LIN {X 0,Y 480.885,Z 595.896,A -85,B 0,C 180,E1 22639.921,E2 22639.921} C_VEL
LIN {X 0,Y 480.883,Z 595.897,A -85,B 0,C 180,E1 22636.346,E2 22636.346} C_VEL
LIN {X 0,Y 480.836,Z 595.897,A -85,B 0,C 180,E1 22632.842,E2 22632.842} C_VEL
LIN {X 0,Y 480.862,Z 595.898,A -85,B 0,C 180,E1 22629.331,E2 22629.331} C_VEL
LIN {X 0,Y 480.868,Z 596.139,A -85,B 0,C 180,E1 22626.726,E2 22626.726} C_VEL
LIN {X 0,Y 487.982,Z 616.092,A -85,B 0,C 180,E1 22624.296,E2 22624.296} C_VEL
LIN {X 0,Y 491.181,Z 625.758,A -85,B 0,C 180,E1 22623.202,E2 22623.202} C_VEL
LIN {X 0,Y 488.684,Z 670.223,A -85,B 0,C 180,E1 22619.477,E2 22619.477} C_VEL
LIN {X 0,Y 487.647,Z 692.767,A -85,B 0,C 180,E1 22617.655,E2 22617.655} C_VEL
LIN {X 0,Y 489.758,Z 709.939,A -85,B 0,C 180,E1 22617.279,E2 22617.279} C_VEL
LIN {X 0,Y 487.922,Z 898.558,A -85,B 0,C 180,E1 22614.449,E2 22614.449} C_VEL
LIN {X 0,Y 487.32,Z 917.588,A -85,B 0,C 180,E1 22613.95,E2 22613.95} C_VEL
LIN {X 0,Y 486.57,Z 936.141,A -85,B 0,C 180,E1 22613.238,E2 22613.238} C_VEL
LIN {X 0,Y 485.716,Z 953.916,A -85,B 0,C 180,E1 22612.33,E2 22612.33} C_VEL
LIN {X 0,Y 484.717,Z 971.45,A -85,B 0,C 180,E1 22611.193,E2 22611.193} C_VEL
LIN {X 0,Y 483.784,Z 987.738,A -85,B 0,C 180,E1 22609.886,E2 22609.886} C_VEL
LIN {X 0,Y 482.865,Z 1003.139,A -85,B 0,C 180,E1 22608.388,E2 22608.388} C_VEL
LIN {X 0,Y 482.045,Z 1017.074,A -85,B 0,C 180,E1 22606.757,E2 22606.757} C_VEL
LIN {X 0,Y 481.368,Z 1029.509,A -85,B 0,C 180,E1 22605.014,E2 22605.014} C_VEL
LIN {X 0,Y 480.819,Z 1040.852,A -85,B 0,C 180,E1 22603.101,E2 22603.101} C_VEL
LIN {X 0,Y 480.43,Z 1050.286,A -85,B 0,C 180,E1 22601.16,E2 22601.16} C_VEL
LIN {X 0,Y 480.175,Z 1058.316,A -85,B 0,C 180,E1 22599.106,E2 22599.106} C_VEL
LIN {X 0,Y 480.025,Z 1064.517,A -85,B 0,C 180,E1 22597.059,E2 22597.059} C_VEL
LIN {X 0,Y 479.944,Z 1069.266,A -85,B 0,C 180,E1 22594.9,E2 22594.9} C_VEL
LIN {X 0,Y 479.92,Z 1072.251,A -85,B 0,C 180,E1 22592.747,E2 22592.747} C_VEL
LIN {X 0,Y 479.918,Z 1073.547,A -85,B 0,C 180,E1 22590.597,E2 22590.597} C_VEL
LIN {X 0,Y 479.919,Z 1073.107,A -85,B 0,C 180,E1 22588.329,E2 22588.329} C_VEL
LIN {X 0,Y 479.933,Z 1070.8,A -85,B 0,C 180,E1 22586.058,E2 22586.058} C_VEL
LIN {X 0,Y 479.981,Z 1066.842,A -85,B 0,C 180,E1 22583.902,E2 22583.902} C_VEL
LIN {X 0,Y 480.102,Z 1061.058,A -85,B 0,C 180,E1 22581.738,E2 22581.738} C_VEL
LIN {X 0,Y 480.326,Z 1053.297,A -85,B 0,C 180,E1 22579.566,E2 22579.566} C_VEL
LIN {X 0,Y 480.68,Z 1043.941,A -85,B 0,C 180,E1 22577.507,E2 22577.507} C_VEL
LIN {X 0,Y 481.187,Z 1033.056,A -85,B 0,C 180,E1 22575.561,E2 22575.561} C_VEL
LIN {X 0,Y 481.832,Z 1020.659,A -85,B 0,C 180,E1 22573.732,E2 22573.732} C_VEL
LIN {X 0,Y 482.639,Z 1006.709,A -85,B 0,C 180,E1 22572.021,E2 22572.021} C_VEL
LIN {X 0,Y 483.522,Z 991.701,A -85,B 0,C 180,E1 22570.491,E2 22570.491} C_VEL
LIN {X 0,Y 484.44,Z 975.717,A -85,B 0,C 180,E1 22569.143,E2 22569.143} C_VEL
LIN {X 0,Y 485.421,Z 958.353,A -85,B 0,C 180,E1 22567.956,E2 22567.956} C_VEL
LIN {X 0,Y 486.296,Z 940.865,A -85,B 0,C 180,E1 22567.005,E2 22567.005} C_VEL
LIN {X 0,Y 487.081,Z 922.417,A -85,B 0,C 180,E1 22566.239,E2 22566.239} C_VEL
LIN {X 0,Y 487.711,Z 903.808,A -85,B 0,C 180,E1 22565.693,E2 22565.693} C_VEL
LIN {X 0,Y 488.08,Z 882.284,A -85,B 0,C 180,E1 22565.306,E2 22565.306} C_VEL
LIN {X 0,Y 489.493,Z 707.074,A -85,B 0,C 180,E1 22562.699,E2 22562.699} C_VEL
LIN {X 0,Y 487.571,Z 692.581,A -85,B 0,C 180,E1 22562.362,E2 22562.362} C_VEL
LIN {X 0,Y 489.651,Z 650.462,A -85,B 0,C 180,E1 22558.894,E2 22558.894} C_VEL
LIN {X 0,Y 491.217,Z 625.654,A -85,B 0,C 180,E1 22556.781,E2 22556.781} C_VEL
LIN {X 0,Y 484.613,Z 606.437,A -85,B 0,C 180,E1 22554.482,E2 22554.482} C_VEL
LIN {X 0,Y 480.883,Z 596.216,A -85,B 0,C 180,E1 22553.128,E2 22553.128} C_VEL
LIN {X 0,Y 480.846,Z 595.905,A -85,B 0,C 180,E1 22551.621,E2 22551.621} C_VEL
LIN {X 0,Y 480.897,Z 595.893,A -85,B 0,C 180,E1 22548.133,E2 22548.133} C_VEL
LIN {X 0,Y 480.845,Z 595.899,A -85,B 0,C 180,E1 22544.654,E2 22544.654} C_VEL
LIN {X 0,Y 480.838,Z 595.9,A -85,B 0,C 180,E1 22541.078,E2 22541.078} C_VEL
LIN {X 0,Y 480.897,Z 595.89,A -85,B 0,C 180,E1 22537.681,E2 22537.681} C_VEL
LIN {X 0,Y 480.854,Z 595.896,A -85,B 0,C 180,E1 22534.149,E2 22534.149} C_VEL
LIN {X 0,Y 480.837,Z 595.9,A -85,B 0,C 180,E1 22530.585,E2 22530.585} C_VEL
LIN {X 0,Y 480.89,Z 595.889,A -85,B 0,C 180,E1 22527.14,E2 22527.14} C_VEL
LIN {X 0,Y 480.863,Z 595.889,A -85,B 0,C 180,E1 22523.66,E2 22523.66} C_VEL
LIN {X 0,Y 480.841,Z 595.894,A -85,B 0,C 180,E1 22520.193,E2 22520.193} C_VEL
LIN {X 0,Y 480.885,Z 595.899,A -85,B 0,C 180,E1 22516.674,E2 22516.674} C_VEL
LIN {X 0,Y 480.867,Z 595.89,A -85,B 0,C 180,E1 22513.222,E2 22513.222} C_VEL
LIN {X 0,Y 480.843,Z 595.886,A -85,B 0,C 180,E1 22509.696,E2 22509.696} C_VEL
LIN {X 0,Y 480.881,Z 595.895,A -85,B 0,C 180,E1 22506.207,E2 22506.207} C_VEL
LIN {X 0,Y 480.882,Z 595.893,A -85,B 0,C 180,E1 22502.622,E2 22502.622} C_VEL
LIN {X 0,Y 480.848,Z 595.892,A -85,B 0,C 180,E1 22499.166,E2 22499.166} C_VEL
LIN {X 0,Y 480.87,Z 595.888,A -85,B 0,C 180,E1 22495.587,E2 22495.587} C_VEL
LIN {X 0,Y 480.896,Z 595.896,A -85,B 0,C 180,E1 22491.992,E2 22491.992} C_VEL
LIN {X 0,Y 480.859,Z 595.897,A -85,B 0,C 180,E1 22488.485,E2 22488.485} C_VEL
LIN {X 0,Y 480.855,Z 595.899,A -85,B 0,C 180,E1 22484.811,E2 22484.811} C_VEL
LIN {X 0,Y 480.892,Z 595.895,A -85,B 0,C 180,E1 22481.325,E2 22481.325} C_VEL
LIN {X 0,Y 480.886,Z 595.895,A -85,B 0,C 180,E1 22477.706,E2 22477.706} C_VEL
LIN {X 0,Y 480.86,Z 595.897,A -85,B 0,C 180,E1 22474.109,E2 22474.109} C_VEL
LIN {X 0,Y 480.875,Z 595.894,A -85,B 0,C 180,E1 22470.476,E2 22470.476} C_VEL
LIN {X 0,Y 480.893,Z 595.897,A -85,B 0,C 180,E1 22466.85,E2 22466.85} C_VEL
LIN {X 0,Y 480.882,Z 595.898,A -85,B 0,C 180,E1 22463.214,E2 22463.214} C_VEL
LIN {X 0,Y 480.94,Z 596.225,A -85,B 0,C 180,E1 22462.577,E2 22462.577} C_VEL
LIN {X 0,Y 485.634,Z 612.199,A -85,B 0,C 180,E1 22459.877,E2 22459.877} C_VEL
LIN {X 0,Y 487.628,Z 620.026,A -85,B 0,C 180,E1 22458.631,E2 22458.631} C_VEL
LIN {X 0,Y 485.867,Z 648.971,A -85,B 0,C 180,E1 22454.807,E2 22454.807} C_VEL
LIN {X 0,Y 484.335,Z 678.124,A -85,B 0,C 180,E1 22451.032,E2 22451.032} C_VEL
LIN {X 0,Y 483.003,Z 708.393,A -85,B 0,C 180,E1 22447.182,E2 22447.182} C_VEL
LIN {X 0,Y 483.679,Z 712.593,A -85,B 0,C 180,E1 22447.023,E2 22447.023} C_VEL
LIN {X 0,Y 484.283,Z 715.766,A -85,B 0,C 180,E1 22446.942,E2 22446.942} C_VEL
LIN {X 0,Y 484.176,Z 720.144,A -85,B 0,C 180,E1 22446.877,E2 22446.877} C_VEL
LIN {X 0,Y 481.662,Z 727.25,A -85,B 0,C 180,E1 22446.89,E2 22446.89} C_VEL
LIN {X 0,Y 478.477,Z 735.14,A -85,B 0,C 180,E1 22446.924,E2 22446.924} C_VEL
LIN {X 0,Y 477.919,Z 738.903,A -85,B 0,C 180,E1 22446.892,E2 22446.892} C_VEL
LIN {X 0,Y 476.905,Z 825.971,A -85,B 0,C 180,E1 22445.471,E2 22445.471} C_VEL
LIN {X 0,Y 476.579,Z 841.641,A -85,B 0,C 180,E1 22444.979,E2 22444.979} C_VEL
LIN {X 0,Y 476.066,Z 856.592,A -85,B 0,C 180,E1 22444.254,E2 22444.254} C_VEL
LIN {X 0,Y 475.466,Z 870.004,A -85,B 0,C 180,E1 22443.361,E2 22443.361} C_VEL
LIN {X 0,Y 474.82,Z 882.624,A -85,B 0,C 180,E1 22442.265,E2 22442.265} C_VEL
LIN {X 0,Y 474.198,Z 894.207,A -85,B 0,C 180,E1 22440.963,E2 22440.963} C_VEL
LIN {X 0,Y 473.624,Z 903.957,A -85,B 0,C 180,E1 22439.568,E2 22439.568} C_VEL
LIN {X 0,Y 473.133,Z 912.641,A -85,B 0,C 180,E1 22437.979,E2 22437.979} C_VEL
LIN {X 0,Y 472.77,Z 919.786,A -85,B 0,C 180,E1 22436.232,E2 22436.232} C_VEL
LIN {X 0,Y 472.546,Z 924.839,A -85,B 0,C 180,E1 22434.501,E2 22434.501} C_VEL
LIN {X 0,Y 472.426,Z 928.327,A -85,B 0,C 180,E1 22432.655,E2 22432.655} C_VEL
LIN {X 0,Y 472.374,Z 930.028,A -85,B 0,C 180,E1 22430.679,E2 22430.679} C_VEL
LIN {X 0,Y 472.37,Z 929.733,A -85,B 0,C 180,E1 22428.768,E2 22428.768} C_VEL
LIN {X 0,Y 472.42,Z 927.698,A -85,B 0,C 180,E1 22426.933,E2 22426.933} C_VEL
LIN {X 0,Y 472.546,Z 923.813,A -85,B 0,C 180,E1 22425.085,E2 22425.085} C_VEL
LIN {X 0,Y 472.773,Z 918.177,A -85,B 0,C 180,E1 22423.328,E2 22423.328} C_VEL
LIN {X 0,Y 473.116,Z 911.095,A -85,B 0,C 180,E1 22421.705,E2 22421.705} C_VEL
LIN {X 0,Y 473.581,Z 902.634,A -85,B 0,C 180,E1 22420.215,E2 22420.215} C_VEL
LIN {X 0,Y 474.15,Z 892.288,A -85,B 0,C 180,E1 22418.794,E2 22418.794} C_VEL
LIN {X 0,Y 474.727,Z 880.939,A -85,B 0,C 180,E1 22417.564,E2 22417.564} C_VEL
LIN {X 0,Y 475.391,Z 867.786,A -85,B 0,C 180,E1 22416.461,E2 22416.461} C_VEL
LIN {X 0,Y 475.944,Z 854.292,A -85,B 0,C 180,E1 22415.606,E2 22415.606} C_VEL
LIN {X 0,Y 476.403,Z 839.891,A -85,B 0,C 180,E1 22414.94,E2 22414.94} C_VEL
LIN {X 0,Y 476.721,Z 823.999,A -85,B 0,C 180,E1 22414.466,E2 22414.466} C_VEL
LIN {X 0,Y 477.568,Z 722.274,A -85,B 0,C 180,E1 22412.847,E2 22412.847} C_VEL
LIN {X 0,Y 475.196,Z 708.93,A -85,B 0,C 180,E1 22412.502,E2 22412.502} C_VEL
LIN {X 0,Y 476.348,Z 681.616,A -85,B 0,C 180,E1 22409.038,E2 22409.038} C_VEL
LIN {X 0,Y 477.85,Z 653.013,A -85,B 0,C 180,E1 22405.319,E2 22405.319} C_VEL
LIN {X 0,Y 479.563,Z 623.964,A -85,B 0,C 180,E1 22401.487,E2 22401.487} C_VEL
LIN {X 0,Y 479.484,Z 620.492,A -85,B 0,C 180,E1 22401.002,E2 22401.002} C_VEL
LIN {X 0,Y 474.295,Z 601.706,A -85,B 0,C 180,E1 22398.004,E2 22398.004} C_VEL
LIN {X 0,Y 472.958,Z 596.977,A -85,B 0,C 180,E1 22397.175,E2 22397.175} C_VEL
LIN {X 0,Y 472.94,Z 596.887,A -85,B 0,C 180,E1 22393.543,E2 22393.543} C_VEL
LIN {X 0,Y 472.936,Z 596.88,A -85,B 0,C 180,E1 22389.833,E2 22389.833} C_VEL
LIN {X 0,Y 472.947,Z 596.853,A -85,B 0,C 180,E1 22386.265,E2 22386.265} C_VEL
LIN {X 0,Y 472.949,Z 596.886,A -85,B 0,C 180,E1 22382.556,E2 22382.556} C_VEL
LIN {X 0,Y 472.931,Z 596.851,A -85,B 0,C 180,E1 22378.945,E2 22378.945} C_VEL
LIN {X 0,Y 472.936,Z 596.883,A -85,B 0,C 180,E1 22375.327,E2 22375.327} C_VEL
LIN {X 0,Y 472.953,Z 596.879,A -85,B 0,C 180,E1 22371.659,E2 22371.659} C_VEL
LIN {X 0,Y 472.949,Z 596.877,A -85,B 0,C 180,E1 22368.082,E2 22368.082} C_VEL
LIN {X 0,Y 472.931,Z 596.885,A -85,B 0,C 180,E1 22364.411,E2 22364.411} C_VEL
LIN {X 0,Y 472.933,Z 596.866,A -85,B 0,C 180,E1 22360.79,E2 22360.79} C_VEL
LIN {X 0,Y 472.952,Z 596.882,A -85,B 0,C 180,E1 22357.202,E2 22357.202} C_VEL
LIN {X 0,Y 472.952,Z 596.869,A -85,B 0,C 180,E1 22353.489,E2 22353.489} C_VEL
LIN {X 0,Y 472.92,Z 596.886,A -85,B 0,C 180,E1 22349.906,E2 22349.906} C_VEL
LIN {X 0,Y 472.934,Z 596.864,A -85,B 0,C 180,E1 22346.309,E2 22346.309} C_VEL
LIN {X 0,Y 472.955,Z 596.884,A -85,B 0,C 180,E1 22342.761,E2 22342.761} C_VEL
LIN {X 0,Y 472.931,Z 596.876,A -85,B 0,C 180,E1 22339.129,E2 22339.129} C_VEL
LIN {X 0,Y 472.916,Z 596.876,A -85,B 0,C 180,E1 22335.576,E2 22335.576} C_VEL
LIN {X 0,Y 472.951,Z 596.878,A -85,B 0,C 180,E1 22332.081,E2 22332.081} C_VEL
LIN {X 0,Y 472.95,Z 596.865,A -85,B 0,C 180,E1 22328.388,E2 22328.388} C_VEL
LIN {X 0,Y 472.913,Z 596.886,A -85,B 0,C 180,E1 22324.852,E2 22324.852} C_VEL
LIN {X 0,Y 472.92,Z 596.867,A -85,B 0,C 180,E1 22321.212,E2 22321.212} C_VEL
LIN {X 0,Y 472.957,Z 596.883,A -85,B 0,C 180,E1 22317.698,E2 22317.698} C_VEL
LIN {X 0,Y 472.919,Z 596.882,A -85,B 0,C 180,E1 22314.176,E2 22314.176} C_VEL
LIN {X 0,Y 472.911,Z 596.881,A -85,B 0,C 180,E1 22310.631,E2 22310.631} C_VEL
LIN {X 0,Y 472.95,Z 596.874,A -85,B 0,C 180,E1 22307.051,E2 22307.051} C_VEL
LIN {X 0,Y 472.949,Z 596.884,A -85,B 0,C 180,E1 22303.417,E2 22303.417} C_VEL
LIN {X 0,Y 472.905,Z 596.882,A -85,B 0,C 180,E1 22299.843,E2 22299.843} C_VEL
LIN {X 0,Y 472.92,Z 596.885,A -85,B 0,C 180,E1 22296.272,E2 22296.272} C_VEL
LIN {X 0,Y 472.96,Z 596.882,A -85,B 0,C 180,E1 22292.694,E2 22292.694} C_VEL
LIN {X 0,Y 472.911,Z 596.883,A -85,B 0,C 180,E1 22289.226,E2 22289.226} C_VEL
LIN {X 0,Y 472.902,Z 596.884,A -85,B 0,C 180,E1 22285.631,E2 22285.631} C_VEL
LIN {X 0,Y 472.958,Z 596.879,A -85,B 0,C 180,E1 22282.188,E2 22282.188} C_VEL
LIN {X 0,Y 472.917,Z 596.888,A -85,B 0,C 180,E1 22278.728,E2 22278.728} C_VEL
LIN {X 0,Y 472.901,Z 596.885,A -85,B 0,C 180,E1 22275.246,E2 22275.246} C_VEL
LIN {X 0,Y 472.958,Z 596.885,A -85,B 0,C 180,E1 22271.733,E2 22271.733} C_VEL
LIN {X 0,Y 472.931,Z 596.887,A -85,B 0,C 180,E1 22268.143,E2 22268.143} C_VEL
LIN {X 0,Y 472.969,Z 597.203,A -85,B 0,C 180,E1 22267.239,E2 22267.239} C_VEL
LIN {X 0,Y 481.529,Z 621.351,A -85,B 0,C 180,E1 22264.268,E2 22264.268} C_VEL
LIN {X 0,Y 483.833,Z 628.63,A -85,B 0,C 180,E1 22263.438,E2 22263.438} C_VEL
LIN {X 0,Y 481.093,Z 673.966,A -85,B 0,C 180,E1 22259.578,E2 22259.578} C_VEL
LIN {X 0,Y 480.128,Z 692.665,A -85,B 0,C 180,E1 22258.031,E2 22258.031} C_VEL
LIN {X 0,Y 482.339,Z 710.927,A -85,B 0,C 180,E1 22257.622,E2 22257.622} C_VEL
LIN {X 0,Y 480.39,Z 897.795,A -85,B 0,C 180,E1 22254.78,E2 22254.78} C_VEL
LIN {X 0,Y 479.761,Z 916.719,A -85,B 0,C 180,E1 22254.279,E2 22254.279} C_VEL
LIN {X 0,Y 478.961,Z 935.157,A -85,B 0,C 180,E1 22253.564,E2 22253.564} C_VEL
LIN {X 0,Y 478.035,Z 953.1,A -85,B 0,C 180,E1 22252.635,E2 22252.635} C_VEL
LIN {X 0,Y 477.002,Z 970.091,A -85,B 0,C 180,E1 22251.52,E2 22251.52} C_VEL
LIN {X 0,Y 475.975,Z 986.913,A -85,B 0,C 180,E1 22250.152,E2 22250.152} C_VEL
LIN {X 0,Y 475.018,Z 1002.004,A -85,B 0,C 180,E1 22248.66,E2 22248.66} C_VEL
LIN {X 0,Y 474.171,Z 1015.629,A -85,B 0,C 180,E1 22247.044,E2 22247.044} C_VEL
LIN {X 0,Y 473.458,Z 1027.902,A -85,B 0,C 180,E1 22245.307,E2 22245.307} C_VEL
LIN {X 0,Y 472.908,Z 1038.859,A -85,B 0,C 180,E1 22243.449,E2 22243.449} C_VEL
LIN {X 0,Y 472.492,Z 1048.46,A -85,B 0,C 180,E1 22241.474,E2 22241.474} C_VEL
LIN {X 0,Y 472.234,Z 1056.686,A -85,B 0,C 180,E1 22239.37,E2 22239.37} C_VEL
LIN {X 0,Y 472.079,Z 1063.293,A -85,B 0,C 180,E1 22237.179,E2 22237.179} C_VEL
LIN {X 0,Y 472.012,Z 1068.061,A -85,B 0,C 180,E1 22234.983,E2 22234.983} C_VEL
LIN {X 0,Y 472.001,Z 1071.059,A -85,B 0,C 180,E1 22232.793,E2 22232.793} C_VEL
LIN {X 0,Y 472.007,Z 1072.358,A -85,B 0,C 180,E1 22230.607,E2 22230.607} C_VEL
LIN {X 0,Y 472.007,Z 1071.984,A -85,B 0,C 180,E1 22228.422,E2 22228.422} C_VEL
LIN {X 0,Y 472.006,Z 1069.929,A -85,B 0,C 180,E1 22226.235,E2 22226.235} C_VEL
LIN {X 0,Y 472.034,Z 1066.147,A -85,B 0,C 180,E1 22224.043,E2 22224.043} C_VEL
LIN {X 0,Y 472.127,Z 1060.917,A -85,B 0,C 180,E1 22221.965,E2 22221.965} C_VEL
LIN {X 0,Y 472.311,Z 1053.855,A -85,B 0,C 180,E1 22219.86,E2 22219.86} C_VEL
LIN {X 0,Y 472.625,Z 1045.012,A -85,B 0,C 180,E1 22217.787,E2 22217.787} C_VEL
LIN {X 0,Y 473.108,Z 1034.601,A -85,B 0,C 180,E1 22215.809,E2 22215.809} C_VEL
LIN {X 0,Y 473.732,Z 1022.735,A -85,B 0,C 180,E1 22213.949,E2 22213.949} C_VEL
LIN {X 0,Y 474.531,Z 1009.398,A -85,B 0,C 180,E1 22212.211,E2 22212.211} C_VEL
LIN {X 0,Y 475.453,Z 994.485,A -85,B 0,C 180,E1 22210.594,E2 22210.594} C_VEL
LIN {X 0,Y 476.443,Z 978.356,A -85,B 0,C 180,E1 22209.149,E2 22209.149} C_VEL
LIN {X 0,Y 477.468,Z 961.529,A -85,B 0,C 180,E1 22207.921,E2 22207.921} C_VEL
LIN {X 0,Y 478.417,Z 944.62,A -85,B 0,C 180,E1 22206.93,E2 22206.93} C_VEL
LIN {X 0,Y 479.245,Z 927.013,A -85,B 0,C 180,E1 22206.125,E2 22206.125} C_VEL
LIN {X 0,Y 479.972,Z 908.387,A -85,B 0,C 180,E1 22205.505,E2 22205.505} C_VEL
LIN {X 0,Y 480.461,Z 889.417,A -85,B 0,C 180,E1 22205.099,E2 22205.099} C_VEL
LIN {X 0,Y 482.093,Z 708.178,A -85,B 0,C 180,E1 22202.357,E2 22202.357} C_VEL
LIN {X 0,Y 480.089,Z 692.742,A -85,B 0,C 180,E1 22201.989,E2 22201.989} C_VEL
LIN {X 0,Y 482.363,Z 651.377,A -85,B 0,C 180,E1 22198.51,E2 22198.51} C_VEL
LIN {X 0,Y 483.943,Z 628.49,A -85,B 0,C 180,E1 22196.52,E2 22196.52} C_VEL
LIN {X 0,Y 477.386,Z 609.08,A -85,B 0,C 180,E1 22194.15,E2 22194.15} C_VEL
LIN {X 0,Y 472.978,Z 597.091,A -85,B 0,C 180,E1 22192.496,E2 22192.496} C_VEL
LIN {X 0,Y 472.893,Z 596.889,A -85,B 0,C 180,E1 22189.195,E2 22189.195} C_VEL
LIN {X 0,Y 472.94,Z 596.887,A -85,B 0,C 180,E1 22185.76,E2 22185.76} C_VEL
LIN {X 0,Y 472.934,Z 596.888,A -85,B 0,C 180,E1 22182.245,E2 22182.245} C_VEL
LIN {X 0,Y 472.893,Z 596.882,A -85,B 0,C 180,E1 22178.744,E2 22178.744} C_VEL
LIN {X 0,Y 472.931,Z 596.881,A -85,B 0,C 180,E1 22175.252,E2 22175.252} C_VEL
LIN {X 0,Y 472.942,Z 596.878,A -85,B 0,C 180,E1 22171.763,E2 22171.763} C_VEL
LIN {X 0,Y 472.898,Z 596.881,A -85,B 0,C 180,E1 22168.269,E2 22168.269} C_VEL
LIN {X 0,Y 472.922,Z 596.884,A -85,B 0,C 180,E1 22164.747,E2 22164.747} C_VEL
LIN {X 0,Y 472.96,Z 596.883,A -85,B 0,C 180,E1 22161.192,E2 22161.192} C_VEL
LIN {X 0,Y 472.912,Z 596.883,A -85,B 0,C 180,E1 22157.598,E2 22157.598} C_VEL
LIN {X 0,Y 472.903,Z 596.881,A -85,B 0,C 180,E1 22153.947,E2 22153.947} C_VEL
LIN {X 0,Y 472.948,Z 596.878,A -85,B 0,C 180,E1 22150.475,E2 22150.475} C_VEL
LIN {X 0,Y 472.948,Z 596.883,A -85,B 0,C 180,E1 22146.799,E2 22146.799} C_VEL
LIN {X 0,Y 472.909,Z 596.885,A -85,B 0,C 180,E1 22143.272,E2 22143.272} C_VEL
LIN {X 0,Y 472.921,Z 596.878,A -85,B 0,C 180,E1 22139.636,E2 22139.636} C_VEL
LIN {X 0,Y 472.952,Z 596.881,A -85,B 0,C 180,E1 22136.121,E2 22136.121} C_VEL
LIN {X 0,Y 472.925,Z 596.885,A -85,B 0,C 180,E1 22132.551,E2 22132.551} C_VEL
LIN {X 0,Y 472.916,Z 596.888,A -85,B 0,C 180,E1 22128.907,E2 22128.907} C_VEL
LIN {X 0,Y 472.947,Z 596.884,A -85,B 0,C 180,E1 22125.304,E2 22125.304} C_VEL
LIN {X 0,Y 472.954,Z 596.879,A -85,B 0,C 180,E1 22121.639,E2 22121.639} C_VEL
LIN {X 0,Y 472.926,Z 596.885,A -85,B 0,C 180,E1 22118.024,E2 22118.024} C_VEL
LIN {X 0,Y 472.922,Z 596.887,A -85,B 0,C 180,E1 22114.315,E2 22114.315} C_VEL
LIN {X 0,Y 472.957,Z 596.881,A -85,B 0,C 180,E1 22110.768,E2 22110.768} C_VEL
LIN {X 0,Y 472.954,Z 596.888,A -85,B 0,C 180,E1 22107.065,E2 22107.065} C_VEL
LIN {X 0,Y 472.933,Z 596.891,A -85,B 0,C 180,E1 22103.402,E2 22103.402} C_VEL
LIN {X 0,Y 473.036,Z 597.438,A -85,B 0,C 180,E1 22103.109,E2 22103.109} C_VEL
LIN {X 0,Y 477.84,Z 613.397,A -85,B 0,C 180,E1 22100.342,E2 22100.342} C_VEL
LIN {X 0,Y 480.223,Z 622.47,A -85,B 0,C 180,E1 22098.857,E2 22098.857} C_VEL
LIN {X 0,Y 478.37,Z 650.86,A -85,B 0,C 180,E1 22095.051,E2 22095.051} C_VEL
LIN {X 0,Y 476.689,Z 680.573,A -85,B 0,C 180,E1 22091.148,E2 22091.148} C_VEL
LIN {X 0,Y 475.403,Z 708.761,A -85,B 0,C 180,E1 22087.542,E2 22087.542} C_VEL
LIN {X 0,Y 478.088,Z 724.621,A -85,B 0,C 180,E1 22087.113,E2 22087.113} C_VEL
LIN {X 0,Y 477.919,Z 738.903,A -85,B 0,C 180,E1 22086.892,E2 22086.892} C_VEL
LIN {X 0,Y 476.895,Z 746.581,A -85,B 0,C 180,E1 22086.819,E2 22086.819} C_VEL
LIN {X 0,Y 470.884,Z 766.961,A -85,B 0,C 180,E1 22086.786,E2 22086.786} C_VEL
LIN {X 0,Y 470.135,Z 773.549,A -85,B 0,C 180,E1 22086.714,E2 22086.714} C_VEL
LIN {X 0,Y 469.431,Z 827.284,A -85,B 0,C 180,E1 22085.795,E2 22085.795} C_VEL
LIN {X 0,Y 469.101,Z 842.121,A -85,B 0,C 180,E1 22085.319,E2 22085.319} C_VEL
LIN {X 0,Y 468.554,Z 857.14,A -85,B 0,C 180,E1 22084.585,E2 22084.585} C_VEL
LIN {X 0,Y 467.962,Z 869.757,A -85,B 0,C 180,E1 22083.747,E2 22083.747} C_VEL
LIN {X 0,Y 467.253,Z 882.637,A -85,B 0,C 180,E1 22082.632,E2 22082.632} C_VEL
LIN {X 0,Y 466.572,Z 894.161,A -85,B 0,C 180,E1 22081.345,E2 22081.345} C_VEL
LIN {X 0,Y 465.975,Z 903.75,A -85,B 0,C 180,E1 22079.997,E2 22079.997} C_VEL
LIN {X 0,Y 465.389,Z 912.872,A -85,B 0,C 180,E1 22078.347,E2 22078.347} C_VEL
LIN {X 0,Y 464.986,Z 919.766,A -85,B 0,C 180,E1 22076.706,E2 22076.706} C_VEL
LIN {X 0,Y 464.714,Z 925.219,A -85,B 0,C 180,E1 22074.942,E2 22074.942} C_VEL
LIN {X 0,Y 464.548,Z 929.014,A -85,B 0,C 180,E1 22073.062,E2 22073.062} C_VEL
LIN {X 0,Y 464.473,Z 930.974,A -85,B 0,C 180,E1 22071.201,E2 22071.201} C_VEL
LIN {X 0,Y 464.457,Z 931.188,A -85,B 0,C 180,E1 22069.23,E2 22069.23} C_VEL
LIN {X 0,Y 464.498,Z 929.472,A -85,B 0,C 180,E1 22067.281,E2 22067.281} C_VEL
LIN {X 0,Y 464.615,Z 926.158,A -85,B 0,C 180,E1 22065.477,E2 22065.477} C_VEL
LIN {X 0,Y 464.84,Z 921.078,A -85,B 0,C 180,E1 22063.686,E2 22063.686} C_VEL
LIN {X 0,Y 465.17,Z 914.536,A -85,B 0,C 180,E1 22062.034,E2 22062.034} C_VEL
LIN {X 0,Y 465.655,Z 906.316,A -85,B 0,C 180,E1 22060.445,E2 22060.445} C_VEL
LIN {X 0,Y 466.294,Z 895.8,A -85,B 0,C 180,E1 22058.881,E2 22058.881} C_VEL
LIN {X 0,Y 466.914,Z 884.437,A -85,B 0,C 180,E1 22057.567,E2 22057.567} C_VEL
LIN {X 0,Y 467.553,Z 872.845,A -85,B 0,C 180,E1 22056.508,E2 22056.508} C_VEL
LIN {X 0,Y 468.223,Z 858.64,A -85,B 0,C 180,E1 22055.514,E2 22055.514} C_VEL
LIN {X 0,Y 468.73,Z 844.762,A -85,B 0,C 180,E1 22054.803,E2 22054.803} C_VEL
LIN {X 0,Y 469.111,Z 829.612,A -85,B 0,C 180,E1 22054.27,E2 22054.27} C_VEL
LIN {X 0,Y 469.364,Z 808.595,A -85,B 0,C 180,E1 22053.868,E2 22053.868} C_VEL
LIN {X 0,Y 470.112,Z 723.231,A -85,B 0,C 180,E1 22052.503,E2 22052.503} C_VEL
LIN {X 0,Y 467.517,Z 708.651,A -85,B 0,C 180,E1 22052.114,E2 22052.114} C_VEL
LIN {X 0,Y 468.86,Z 679.98,A -85,B 0,C 180,E1 22048.411,E2 22048.411} C_VEL
LIN {X 0,Y 470.534,Z 650.401,A -85,B 0,C 180,E1 22044.513,E2 22044.513} C_VEL
LIN {X 0,Y 472.212,Z 623.861,A -85,B 0,C 180,E1 22040.954,E2 22040.954} C_VEL
LIN {X 0,Y 467.015,Z 604.886,A -85,B 0,C 180,E1 22037.888,E2 22037.888} C_VEL
LIN {X 0,Y 465.024,Z 597.986,A -85,B 0,C 180,E1 22036.699,E2 22036.699} C_VEL
LIN {X 0,Y 465.01,Z 597.873,A -85,B 0,C 180,E1 22032.996,E2 22032.996} C_VEL
LIN {X 0,Y 465.005,Z 597.872,A -85,B 0,C 180,E1 22029.284,E2 22029.284} C_VEL
LIN {X 0,Y 464.992,Z 597.843,A -85,B 0,C 180,E1 22025.615,E2 22025.615} C_VEL
LIN {X 0,Y 465.014,Z 597.869,A -85,B 0,C 180,E1 22021.908,E2 22021.908} C_VEL
LIN {X 0,Y 465.007,Z 597.843,A -85,B 0,C 180,E1 22018.21,E2 22018.21} C_VEL
LIN {X 0,Y 465.006,Z 597.878,A -85,B 0,C 180,E1 22014.51,E2 22014.51} C_VEL
LIN {X 0,Y 464.99,Z 597.871,A -85,B 0,C 180,E1 22010.919,E2 22010.919} C_VEL
LIN {X 0,Y 465.007,Z 597.858,A -85,B 0,C 180,E1 22007.339,E2 22007.339} C_VEL
LIN {X 0,Y 465.013,Z 597.872,A -85,B 0,C 180,E1 22003.647,E2 22003.647} C_VEL
LIN {X 0,Y 465,Z 597.859,A -85,B 0,C 180,E1 22000.01,E2 22000.01} C_VEL
LIN {X 0,Y 464.988,Z 597.872,A -85,B 0,C 180,E1 21996.405,E2 21996.405} C_VEL
LIN {X 0,Y 465.01,Z 597.861,A -85,B 0,C 180,E1 21992.782,E2 21992.782} C_VEL
LIN {X 0,Y 465.017,Z 597.87,A -85,B 0,C 180,E1 21989.074,E2 21989.074} C_VEL
LIN {X 0,Y 464.991,Z 597.855,A -85,B 0,C 180,E1 21985.428,E2 21985.428} C_VEL
LIN {X 0,Y 464.981,Z 597.873,A -85,B 0,C 180,E1 21981.84,E2 21981.84} C_VEL
LIN {X 0,Y 465.01,Z 597.85,A -85,B 0,C 180,E1 21978.296,E2 21978.296} C_VEL
LIN {X 0,Y 465.021,Z 597.873,A -85,B 0,C 180,E1 21974.571,E2 21974.571} C_VEL
LIN {X 0,Y 464.983,Z 597.87,A -85,B 0,C 180,E1 21970.908,E2 21970.908} C_VEL
LIN {X 0,Y 464.976,Z 597.862,A -85,B 0,C 180,E1 21967.289,E2 21967.289} C_VEL
LIN {X 0,Y 465.009,Z 597.867,A -85,B 0,C 180,E1 21963.699,E2 21963.699} C_VEL
LIN {X 0,Y 465.019,Z 597.854,A -85,B 0,C 180,E1 21960,E2 21960} C_VEL
LIN {X 0,Y 464.973,Z 597.877,A -85,B 0,C 180,E1 21956.425,E2 21956.425} C_VEL
LIN {X 0,Y 464.971,Z 597.856,A -85,B 0,C 180,E1 21952.711,E2 21952.711} C_VEL
LIN {X 0,Y 465.013,Z 597.872,A -85,B 0,C 180,E1 21949.219,E2 21949.219} C_VEL
LIN {X 0,Y 465.004,Z 597.86,A -85,B 0,C 180,E1 21945.557,E2 21945.557} C_VEL
LIN {X 0,Y 464.965,Z 597.877,A -85,B 0,C 180,E1 21942.091,E2 21942.091} C_VEL
LIN {X 0,Y 464.997,Z 597.866,A -85,B 0,C 180,E1 21938.559,E2 21938.559} C_VEL
LIN {X 0,Y 465.015,Z 597.865,A -85,B 0,C 180,E1 21934.939,E2 21934.939} C_VEL
LIN {X 0,Y 464.965,Z 597.878,A -85,B 0,C 180,E1 21931.485,E2 21931.485} C_VEL
LIN {X 0,Y 464.977,Z 597.873,A -85,B 0,C 180,E1 21927.913,E2 21927.913} C_VEL
LIN {X 0,Y 465.016,Z 597.87,A -85,B 0,C 180,E1 21924.36,E2 21924.36} C_VEL
LIN {X 0,Y 464.979,Z 597.872,A -85,B 0,C 180,E1 21920.788,E2 21920.788} C_VEL
LIN {X 0,Y 464.959,Z 597.878,A -85,B 0,C 180,E1 21917.193,E2 21917.193} C_VEL
LIN {X 0,Y 465,Z 597.872,A -85,B 0,C 180,E1 21913.649,E2 21913.649} C_VEL
LIN {X 0,Y 465.014,Z 597.874,A -85,B 0,C 180,E1 21910.009,E2 21910.009} C_VEL
LIN {X 0,Y 465.049,Z 598.088,A -85,B 0,C 180,E1 21907.816,E2 21907.816} C_VEL
LIN {X 0,Y 473.531,Z 622.006,A -85,B 0,C 180,E1 21904.778,E2 21904.778} C_VEL
LIN {X 0,Y 476.501,Z 630.993,A -85,B 0,C 180,E1 21903.719,E2 21903.719} C_VEL
LIN {X 0,Y 473.525,Z 676.833,A -85,B 0,C 180,E1 21899.75,E2 21899.75} C_VEL
LIN {X 0,Y 472.663,Z 693.247,A -85,B 0,C 180,E1 21898.388,E2 21898.388} C_VEL
LIN {X 0,Y 474.919,Z 711.941,A -85,B 0,C 180,E1 21897.969,E2 21897.969} C_VEL
LIN {X 0,Y 472.863,Z 897.281,A -85,B 0,C 180,E1 21895.114,E2 21895.114} C_VEL
LIN {X 0,Y 472.198,Z 916.282,A -85,B 0,C 180,E1 21894.602,E2 21894.602} C_VEL
LIN {X 0,Y 471.368,Z 934.175,A -85,B 0,C 180,E1 21893.901,E2 21893.901} C_VEL
LIN {X 0,Y 470.444,Z 951.114,A -85,B 0,C 180,E1 21893.021,E2 21893.021} C_VEL
LIN {X 0,Y 469.343,Z 968.315,A -85,B 0,C 180,E1 21891.889,E2 21891.889} C_VEL
LIN {X 0,Y 468.281,Z 984.589,A -85,B 0,C 180,E1 21890.563,E2 21890.563} C_VEL
LIN {X 0,Y 467.249,Z 999.901,A -85,B 0,C 180,E1 21889.047,E2 21889.047} C_VEL
LIN {X 0,Y 466.305,Z 1014.184,A -85,B 0,C 180,E1 21887.341,E2 21887.341} C_VEL
LIN {X 0,Y 465.5,Z 1027.329,A -85,B 0,C 180,E1 21885.447,E2 21885.447} C_VEL
LIN {X 0,Y 464.935,Z 1038.197,A -85,B 0,C 180,E1 21883.557,E2 21883.557} C_VEL
LIN {X 0,Y 464.516,Z 1047.716,A -85,B 0,C 180,E1 21881.548,E2 21881.548} C_VEL
LIN {X 0,Y 464.266,Z 1055.816,A -85,B 0,C 180,E1 21879.421,E2 21879.421} C_VEL
LIN {X 0,Y 464.132,Z 1062.068,A -85,B 0,C 180,E1 21877.302,E2 21877.302} C_VEL
LIN {X 0,Y 464.08,Z 1066.856,A -85,B 0,C 180,E1 21875.068,E2 21875.068} C_VEL
LIN {X 0,Y 464.083,Z 1069.865,A -85,B 0,C 180,E1 21872.841,E2 21872.841} C_VEL
LIN {X 0,Y 464.096,Z 1071.167,A -85,B 0,C 180,E1 21870.617,E2 21870.617} C_VEL
LIN {X 0,Y 464.094,Z 1070.787,A -85,B 0,C 180,E1 21868.395,E2 21868.395} C_VEL
LIN {X 0,Y 464.085,Z 1068.717,A -85,B 0,C 180,E1 21866.171,E2 21866.171} C_VEL
LIN {X 0,Y 464.101,Z 1064.912,A -85,B 0,C 180,E1 21863.94,E2 21863.94} C_VEL
LIN {X 0,Y 464.178,Z 1059.65,A -85,B 0,C 180,E1 21861.827,E2 21861.827} C_VEL
LIN {X 0,Y 464.352,Z 1052.63,A -85,B 0,C 180,E1 21859.705,E2 21859.705} C_VEL
LIN {X 0,Y 464.678,Z 1043.661,A -85,B 0,C 180,E1 21857.575,E2 21857.575} C_VEL
LIN {X 0,Y 465.179,Z 1033.193,A -85,B 0,C 180,E1 21855.562,E2 21855.562} C_VEL
LIN {X 0,Y 465.839,Z 1021.26,A -85,B 0,C 180,E1 21853.67,E2 21853.67} C_VEL
LIN {X 0,Y 466.688,Z 1007.842,A -85,B 0,C 180,E1 21851.901,E2 21851.901} C_VEL
LIN {X 0,Y 467.673,Z 992.825,A -85,B 0,C 180,E1 21850.258,E2 21850.258} C_VEL
LIN {X 0,Y 468.728,Z 976.645,A -85,B 0,C 180,E1 21848.797,E2 21848.797} C_VEL
LIN {X 0,Y 469.818,Z 959.856,A -85,B 0,C 180,E1 21847.564,E2 21847.564} C_VEL
LIN {X 0,Y 470.834,Z 942.582,A -85,B 0,C 180,E1 21846.548,E2 21846.548} C_VEL
LIN {X 0,Y 471.717,Z 925.142,A -85,B 0,C 180,E1 21845.753,E2 21845.753} C_VEL
LIN {X 0,Y 472.481,Z 906.497,A -85,B 0,C 180,E1 21845.136,E2 21845.136} C_VEL
LIN {X 0,Y 472.976,Z 887.127,A -85,B 0,C 180,E1 21844.731,E2 21844.731} C_VEL
LIN {X 0,Y 474.685,Z 709.08,A -85,B 0,C 180,E1 21841.998,E2 21841.998} C_VEL
LIN {X 0,Y 472.632,Z 693.093,A -85,B 0,C 180,E1 21841.614,E2 21841.614} C_VEL
LIN {X 0,Y 474.934,Z 654.519,A -85,B 0,C 180,E1 21838.307,E2 21838.307} C_VEL
LIN {X 0,Y 476.533,Z 630.773,A -85,B 0,C 180,E1 21836.19,E2 21836.19} C_VEL
LIN {X 0,Y 470.34,Z 612.376,A -85,B 0,C 180,E1 21833.882,E2 21833.882} C_VEL
LIN {X 0,Y 465.025,Z 598.126,A -85,B 0,C 180,E1 21831.861,E2 21831.861} C_VEL
LIN {X 0,Y 464.977,Z 597.873,A -85,B 0,C 180,E1 21828.631,E2 21828.631} C_VEL
LIN {X 0,Y 464.957,Z 597.88,A -85,B 0,C 180,E1 21825.143,E2 21825.143} C_VEL
LIN {X 0,Y 465.006,Z 597.87,A -85,B 0,C 180,E1 21821.637,E2 21821.637} C_VEL
LIN {X 0,Y 464.995,Z 597.866,A -85,B 0,C 180,E1 21818.094,E2 21818.094} C_VEL
LIN {X 0,Y 464.959,Z 597.876,A -85,B 0,C 180,E1 21814.552,E2 21814.552} C_VEL
LIN {X 0,Y 464.987,Z 597.87,A -85,B 0,C 180,E1 21811.069,E2 21811.069} C_VEL
LIN {X 0,Y 465.01,Z 597.863,A -85,B 0,C 180,E1 21807.535,E2 21807.535} C_VEL
LIN {X 0,Y 464.966,Z 597.868,A -85,B 0,C 180,E1 21803.948,E2 21803.948} C_VEL
LIN {X 0,Y 464.965,Z 597.872,A -85,B 0,C 180,E1 21800.256,E2 21800.256} C_VEL
LIN {X 0,Y 465.012,Z 597.875,A -85,B 0,C 180,E1 21796.745,E2 21796.745} C_VEL
LIN {X 0,Y 464.993,Z 597.867,A -85,B 0,C 180,E1 21793.175,E2 21793.175} C_VEL
LIN {X 0,Y 464.967,Z 597.862,A -85,B 0,C 180,E1 21789.656,E2 21789.656} C_VEL
LIN {X 0,Y 464.989,Z 597.871,A -85,B 0,C 180,E1 21786.048,E2 21786.048} C_VEL
LIN {X 0,Y 465.012,Z 597.872,A -85,B 0,C 180,E1 21782.464,E2 21782.464} C_VEL
LIN {X 0,Y 464.978,Z 597.869,A -85,B 0,C 180,E1 21778.891,E2 21778.891} C_VEL
LIN {X 0,Y 464.973,Z 597.865,A -85,B 0,C 180,E1 21775.189,E2 21775.189} C_VEL
LIN {X 0,Y 465.007,Z 597.866,A -85,B 0,C 180,E1 21771.592,E2 21771.592} C_VEL
LIN {X 0,Y 465.011,Z 597.874,A -85,B 0,C 180,E1 21767.961,E2 21767.961} C_VEL
LIN {X 0,Y 464.979,Z 597.875,A -85,B 0,C 180,E1 21764.407,E2 21764.407} C_VEL
LIN {X 0,Y 464.982,Z 597.876,A -85,B 0,C 180,E1 21760.661,E2 21760.661} C_VEL
LIN {X 0,Y 465.015,Z 597.873,A -85,B 0,C 180,E1 21757.096,E2 21757.096} C_VEL
LIN {X 0,Y 465.013,Z 597.87,A -85,B 0,C 180,E1 21753.433,E2 21753.433} C_VEL
LIN {X 0,Y 464.985,Z 597.876,A -85,B 0,C 180,E1 21749.817,E2 21749.817} C_VEL
LIN {X 0,Y 464.99,Z 597.874,A -85,B 0,C 180,E1 21746.1,E2 21746.1} C_VEL
LIN {X 0,Y 465.02,Z 598.121,A -85,B 0,C 180,E1 21743.788,E2 21743.788} C_VEL
LIN {X 0,Y 469.634,Z 613.048,A -85,B 0,C 180,E1 21741.092,E2 21741.092} C_VEL
LIN {X 0,Y 472.825,Z 625.469,A -85,B 0,C 180,E1 21739.019,E2 21739.019} C_VEL
LIN {X 0,Y 470.747,Z 654.916,A -85,B 0,C 180,E1 21735.015,E2 21735.015} C_VEL
LIN {X 0,Y 469.02,Z 683.674,A -85,B 0,C 180,E1 21731.19,E2 21731.19} C_VEL
LIN {X 0,Y 467.796,Z 708.566,A -85,B 0,C 180,E1 21727.958,E2 21727.958} C_VEL
LIN {X 0,Y 470.722,Z 725.738,A -85,B 0,C 180,E1 21727.479,E2 21727.479} C_VEL
LIN {X 0,Y 470.135,Z 773.549,A -85,B 0,C 180,E1 21726.714,E2 21726.714} C_VEL
LIN {X 0,Y 469.136,Z 781.223,A -85,B 0,C 180,E1 21726.636,E2 21726.636} C_VEL
LIN {X 0,Y 463.045,Z 801.586,A -85,B 0,C 180,E1 21726.594,E2 21726.594} C_VEL
LIN {X 0,Y 462.265,Z 808.171,A -85,B 0,C 180,E1 21726.517,E2 21726.517} C_VEL
LIN {X 0,Y 461.94,Z 830.417,A -85,B 0,C 180,E1 21726.082,E2 21726.082} C_VEL
LIN {X 0,Y 461.554,Z 845.034,A -85,B 0,C 180,E1 21725.567,E2 21725.567} C_VEL
LIN {X 0,Y 461.006,Z 858.927,A -85,B 0,C 180,E1 21724.855,E2 21724.855} C_VEL
LIN {X 0,Y 460.314,Z 872.271,A -85,B 0,C 180,E1 21723.926,E2 21723.926} C_VEL
LIN {X 0,Y 459.572,Z 884.747,A -85,B 0,C 180,E1 21722.802,E2 21722.802} C_VEL
LIN {X 0,Y 458.804,Z 896.852,A -85,B 0,C 180,E1 21721.389,E2 21721.389} C_VEL
LIN {X 0,Y 458.127,Z 906.468,A -85,B 0,C 180,E1 21719.951,E2 21719.951} C_VEL
LIN {X 0,Y 457.535,Z 915.078,A -85,B 0,C 180,E1 21718.308,E2 21718.308} C_VEL
LIN {X 0,Y 457.085,Z 922.184,A -85,B 0,C 180,E1 21716.503,E2 21716.503} C_VEL
LIN {X 0,Y 456.797,Z 927.213,A -85,B 0,C 180,E1 21714.713,E2 21714.713} C_VEL
LIN {X 0,Y 456.633,Z 930.699,A -85,B 0,C 180,E1 21712.803,E2 21712.803} C_VEL
LIN {X 0,Y 456.557,Z 932.407,A -85,B 0,C 180,E1 21710.75,E2 21710.75} C_VEL
LIN {X 0,Y 456.55,Z 932.14,A -85,B 0,C 180,E1 21708.78,E2 21708.78} C_VEL
LIN {X 0,Y 456.616,Z 930.157,A -85,B 0,C 180,E1 21706.88,E2 21706.88} C_VEL
LIN {X 0,Y 456.772,Z 926.321,A -85,B 0,C 180,E1 21704.969,E2 21704.969} C_VEL
LIN {X 0,Y 457.051,Z 920.775,A -85,B 0,C 180,E1 21703.151,E2 21703.151} C_VEL
LIN {X 0,Y 457.462,Z 913.818,A -85,B 0,C 180,E1 21701.472,E2 21701.472} C_VEL
LIN {X 0,Y 458.05,Z 904.685,A -85,B 0,C 180,E1 21699.803,E2 21699.803} C_VEL
LIN {X 0,Y 458.685,Z 894.826,A -85,B 0,C 180,E1 21698.398,E2 21698.398} C_VEL
LIN {X 0,Y 459.352,Z 883.624,A -85,B 0,C 180,E1 21697.127,E2 21697.127} C_VEL
LIN {X 0,Y 460.093,Z 870.661,A -85,B 0,C 180,E1 21695.987,E2 21695.987} C_VEL
LIN {X 0,Y 460.745,Z 857.103,A -85,B 0,C 180,E1 21695.076,E2 21695.076} C_VEL
LIN {X 0,Y 461.296,Z 842.339,A -85,B 0,C 180,E1 21694.351,E2 21694.351} C_VEL
LIN {X 0,Y 461.657,Z 826.326,A -85,B 0,C 180,E1 21693.842,E2 21693.842} C_VEL
LIN {X 0,Y 462.7,Z 724.376,A -85,B 0,C 180,E1 21692.152,E2 21692.152} C_VEL
LIN {X 0,Y 459.894,Z 708.848,A -85,B 0,C 180,E1 21691.744,E2 21691.744} C_VEL
LIN {X 0,Y 460.105,Z 702.741,A -85,B 0,C 180,E1 21690.996,E2 21690.996} C_VEL
LIN {X 0,Y 461.725,Z 672.697,A -85,B 0,C 180,E1 21687.021,E2 21687.021} C_VEL
LIN {X 0,Y 463.501,Z 644.089,A -85,B 0,C 180,E1 21683.186,E2 21683.186} C_VEL
LIN {X 0,Y 464.619,Z 625.965,A -85,B 0,C 180,E1 21680.712,E2 21680.712} C_VEL
LIN {X 0,Y 459.541,Z 607.471,A -85,B 0,C 180,E1 21677.669,E2 21677.669} C_VEL
LIN {X 0,Y 457.078,Z 598.958,A -85,B 0,C 180,E1 21676.173,E2 21676.173} C_VEL
LIN {X 0,Y 457.072,Z 598.858,A -85,B 0,C 180,E1 21672.429,E2 21672.429} C_VEL
LIN {X 0,Y 457.07,Z 598.864,A -85,B 0,C 180,E1 21668.707,E2 21668.707} C_VEL
LIN {X 0,Y 457.062,Z 598.837,A -85,B 0,C 180,E1 21665.026,E2 21665.026} C_VEL
LIN {X 0,Y 457.055,Z 598.856,A -85,B 0,C 180,E1 21661.311,E2 21661.311} C_VEL
LIN {X 0,Y 457.064,Z 598.842,A -85,B 0,C 180,E1 21657.591,E2 21657.591} C_VEL
LIN {X 0,Y 457.072,Z 598.858,A -85,B 0,C 180,E1 21653.953,E2 21653.953} C_VEL
LIN {X 0,Y 457.077,Z 598.866,A -85,B 0,C 180,E1 21650.159,E2 21650.159} C_VEL
LIN {X 0,Y 457.056,Z 598.85,A -85,B 0,C 180,E1 21646.394,E2 21646.394} C_VEL
LIN {X 0,Y 457.051,Z 598.86,A -85,B 0,C 180,E1 21642.688,E2 21642.688} C_VEL
LIN {X 0,Y 457.08,Z 598.855,A -85,B 0,C 180,E1 21639.05,E2 21639.05} C_VEL
LIN {X 0,Y 457.073,Z 598.849,A -85,B 0,C 180,E1 21635.276,E2 21635.276} C_VEL
LIN {X 0,Y 457.057,Z 598.857,A -85,B 0,C 180,E1 21631.67,E2 21631.67} C_VEL
LIN {X 0,Y 457.045,Z 598.859,A -85,B 0,C 180,E1 21628.057,E2 21628.057} C_VEL
LIN {X 0,Y 457.067,Z 598.851,A -85,B 0,C 180,E1 21624.422,E2 21624.422} C_VEL
LIN {X 0,Y 457.077,Z 598.858,A -85,B 0,C 180,E1 21620.756,E2 21620.756} C_VEL
LIN {X 0,Y 457.05,Z 598.841,A -85,B 0,C 180,E1 21617.047,E2 21617.047} C_VEL
LIN {X 0,Y 457.039,Z 598.863,A -85,B 0,C 180,E1 21613.409,E2 21613.409} C_VEL
LIN {X 0,Y 457.062,Z 598.841,A -85,B 0,C 180,E1 21609.825,E2 21609.825} C_VEL
LIN {X 0,Y 457.08,Z 598.86,A -85,B 0,C 180,E1 21606.153,E2 21606.153} C_VEL
LIN {X 0,Y 457.045,Z 598.858,A -85,B 0,C 180,E1 21602.508,E2 21602.508} C_VEL
LIN {X 0,Y 457.032,Z 598.854,A -85,B 0,C 180,E1 21598.852,E2 21598.852} C_VEL
LIN {X 0,Y 457.062,Z 598.857,A -85,B 0,C 180,E1 21595.232,E2 21595.232} C_VEL
LIN {X 0,Y 457.079,Z 598.849,A -85,B 0,C 180,E1 21591.572,E2 21591.572} C_VEL
LIN {X 0,Y 457.04,Z 598.868,A -85,B 0,C 180,E1 21587.933,E2 21587.933} C_VEL
LIN {X 0,Y 457.028,Z 598.856,A -85,B 0,C 180,E1 21584.284,E2 21584.284} C_VEL
LIN {X 0,Y 457.064,Z 598.855,A -85,B 0,C 180,E1 21580.712,E2 21580.712} C_VEL
LIN {X 0,Y 457.082,Z 598.863,A -85,B 0,C 180,E1 21577.064,E2 21577.064} C_VEL
LIN {X 0,Y 457.03,Z 598.854,A -85,B 0,C 180,E1 21573.482,E2 21573.482} C_VEL
LIN {X 0,Y 457.028,Z 598.86,A -85,B 0,C 180,E1 21569.788,E2 21569.788} C_VEL
LIN {X 0,Y 457.069,Z 598.858,A -85,B 0,C 180,E1 21566.23,E2 21566.23} C_VEL
LIN {X 0,Y 457.069,Z 598.862,A -85,B 0,C 180,E1 21562.545,E2 21562.545} C_VEL
LIN {X 0,Y 457.022,Z 598.87,A -85,B 0,C 180,E1 21559.007,E2 21559.007} C_VEL
LIN {X 0,Y 457.027,Z 598.861,A -85,B 0,C 180,E1 21555.318,E2 21555.318} C_VEL
LIN {X 0,Y 457.082,Z 598.863,A -85,B 0,C 180,E1 21551.761,E2 21551.761} C_VEL
LIN {X 0,Y 457.061,Z 599.078,A -85,B 0,C 180,E1 21548.38,E2 21548.38} C_VEL
LIN {X 0,Y 463.48,Z 617.048,A -85,B 0,C 180,E1 21546.004,E2 21546.004} C_VEL
LIN {X 0,Y 469.14,Z 633.78,A -85,B 0,C 180,E1 21543.967,E2 21543.967} C_VEL
LIN {X 0,Y 465.932,Z 680.105,A -85,B 0,C 180,E1 21539.893,E2 21539.893} C_VEL
LIN {X 0,Y 465.198,Z 693.467,A -85,B 0,C 180,E1 21538.772,E2 21538.772} C_VEL
LIN {X 0,Y 467.52,Z 712.976,A -85,B 0,C 180,E1 21538.328,E2 21538.328} C_VEL
LIN {X 0,Y 465.341,Z 896.677,A -85,B 0,C 180,E1 21535.455,E2 21535.455} C_VEL
LIN {X 0,Y 464.641,Z 915.632,A -85,B 0,C 180,E1 21534.937,E2 21534.937} C_VEL
LIN {X 0,Y 463.746,Z 933.726,A -85,B 0,C 180,E1 21534.216,E2 21534.216} C_VEL
LIN {X 0,Y 462.737,Z 951.118,A -85,B 0,C 180,E1 21533.292,E2 21533.292} C_VEL
LIN {X 0,Y 461.583,Z 968.186,A -85,B 0,C 180,E1 21532.143,E2 21532.143} C_VEL
LIN {X 0,Y 460.411,Z 985.038,A -85,B 0,C 180,E1 21530.731,E2 21530.731} C_VEL
LIN {X 0,Y 459.333,Z 1000.11,A -85,B 0,C 180,E1 21529.19,E2 21529.19} C_VEL
LIN {X 0,Y 458.385,Z 1013.708,A -85,B 0,C 180,E1 21527.519,E2 21527.519} C_VEL
LIN {X 0,Y 457.593,Z 1025.948,A -85,B 0,C 180,E1 21525.721,E2 21525.721} C_VEL
LIN {X 0,Y 456.975,Z 1037.273,A -85,B 0,C 180,E1 21523.72,E2 21523.72} C_VEL
LIN {X 0,Y 456.537,Z 1046.971,A -85,B 0,C 180,E1 21521.624,E2 21521.624} C_VEL
LIN {X 0,Y 456.298,Z 1054.991,A -85,B 0,C 180,E1 21519.459,E2 21519.459} C_VEL
LIN {X 0,Y 456.179,Z 1061.164,A -85,B 0,C 180,E1 21517.304,E2 21517.304} C_VEL
LIN {X 0,Y 456.147,Z 1065.87,A -85,B 0,C 180,E1 21515.03,E2 21515.03} C_VEL
LIN {X 0,Y 456.164,Z 1068.791,A -85,B 0,C 180,E1 21512.764,E2 21512.764} C_VEL
LIN {X 0,Y 456.184,Z 1069.999,A -85,B 0,C 180,E1 21510.503,E2 21510.503} C_VEL
LIN {X 0,Y 456.181,Z 1069.516,A -85,B 0,C 180,E1 21508.242,E2 21508.242} C_VEL
LIN {X 0,Y 456.165,Z 1067.333,A -85,B 0,C 180,E1 21505.978,E2 21505.978} C_VEL
LIN {X 0,Y 456.173,Z 1063.405,A -85,B 0,C 180,E1 21503.708,E2 21503.708} C_VEL
LIN {X 0,Y 456.255,Z 1057.632,A -85,B 0,C 180,E1 21501.43,E2 21501.43} C_VEL
LIN {X 0,Y 456.442,Z 1049.862,A -85,B 0,C 180,E1 21499.141,E2 21499.141} C_VEL
LIN {X 0,Y 456.81,Z 1040.486,A -85,B 0,C 180,E1 21496.971,E2 21496.971} C_VEL
LIN {X 0,Y 457.37,Z 1029.565,A -85,B 0,C 180,E1 21494.921,E2 21494.921} C_VEL
LIN {X 0,Y 458.124,Z 1017.118,A -85,B 0,C 180,E1 21492.995,E2 21492.995} C_VEL
LIN {X 0,Y 459.077,Z 1003.096,A -85,B 0,C 180,E1 21491.196,E2 21491.196} C_VEL
LIN {X 0,Y 460.148,Z 987.893,A -85,B 0,C 180,E1 21489.58,E2 21489.58} C_VEL
LIN {X 0,Y 461.27,Z 971.579,A -85,B 0,C 180,E1 21488.158,E2 21488.158} C_VEL
LIN {X 0,Y 462.439,Z 954.639,A -85,B 0,C 180,E1 21486.962,E2 21486.962} C_VEL
LIN {X 0,Y 463.498,Z 936.792,A -85,B 0,C 180,E1 21485.964,E2 21485.964} C_VEL
LIN {X 0,Y 464.427,Z 918.37,A -85,B 0,C 180,E1 21485.186,E2 21485.186} C_VEL
LIN {X 0,Y 465.203,Z 898.839,A -85,B 0,C 180,E1 21484.618,E2 21484.618} C_VEL
LIN {X 0,Y 465.651,Z 870.024,A -85,B 0,C 180,E1 21484.128,E2 21484.128} C_VEL
LIN {X 0,Y 467.318,Z 710.125,A -85,B 0,C 180,E1 21481.631,E2 21481.631} C_VEL
LIN {X 0,Y 465.182,Z 692.986,A -85,B 0,C 180,E1 21481.201,E2 21481.201} C_VEL
LIN {X 0,Y 468.113,Z 650.194,A -85,B 0,C 180,E1 21477.435,E2 21477.435} C_VEL
LIN {X 0,Y 469.294,Z 633.643,A -85,B 0,C 180,E1 21475.921,E2 21475.921} C_VEL
LIN {X 0,Y 463.125,Z 615.11,A -85,B 0,C 180,E1 21473.533,E2 21473.533} C_VEL
LIN {X 0,Y 457.957,Z 601.749,A -85,B 0,C 180,E1 21471.61,E2 21471.61} C_VEL
LIN {X 0,Y 457.041,Z 599.047,A -85,B 0,C 180,E1 21471.152,E2 21471.152} C_VEL
LIN {X 0,Y 457.06,Z 598.867,A -85,B 0,C 180,E1 21467.81,E2 21467.81} C_VEL
LIN {X 0,Y 457.07,Z 598.858,A -85,B 0,C 180,E1 21464.15,E2 21464.15} C_VEL
LIN {X 0,Y 457.024,Z 598.867,A -85,B 0,C 180,E1 21460.61,E2 21460.61} C_VEL
LIN {X 0,Y 457.026,Z 598.869,A -85,B 0,C 180,E1 21456.987,E2 21456.987} C_VEL
LIN {X 0,Y 457.077,Z 598.864,A -85,B 0,C 180,E1 21453.453,E2 21453.453} C_VEL
LIN {X 0,Y 457.058,Z 598.863,A -85,B 0,C 180,E1 21449.774,E2 21449.774} C_VEL
LIN {X 0,Y 457.024,Z 598.866,A -85,B 0,C 180,E1 21446.227,E2 21446.227} C_VEL
LIN {X 0,Y 457.037,Z 598.861,A -85,B 0,C 180,E1 21442.6,E2 21442.6} C_VEL
LIN {X 0,Y 457.077,Z 598.85,A -85,B 0,C 180,E1 21439.022,E2 21439.022} C_VEL
LIN {X 0,Y 457.047,Z 598.86,A -85,B 0,C 180,E1 21435.349,E2 21435.349} C_VEL
LIN {X 0,Y 457.026,Z 598.866,A -85,B 0,C 180,E1 21431.739,E2 21431.739} C_VEL
LIN {X 0,Y 457.055,Z 598.859,A -85,B 0,C 180,E1 21428.175,E2 21428.175} C_VEL
LIN {X 0,Y 457.067,Z 598.849,A -85,B 0,C 180,E1 21424.642,E2 21424.642} C_VEL
LIN {X 0,Y 457.037,Z 598.861,A -85,B 0,C 180,E1 21421.003,E2 21421.003} C_VEL
LIN {X 0,Y 457.034,Z 598.865,A -85,B 0,C 180,E1 21417.241,E2 21417.241} C_VEL
LIN {X 0,Y 457.061,Z 598.863,A -85,B 0,C 180,E1 21413.594,E2 21413.594} C_VEL
LIN {X 0,Y 457.075,Z 598.851,A -85,B 0,C 180,E1 21409.921,E2 21409.921} C_VEL
LIN {X 0,Y 457.054,Z 598.851,A -85,B 0,C 180,E1 21406.205,E2 21406.205} C_VEL
LIN {X 0,Y 457.039,Z 598.857,A -85,B 0,C 180,E1 21402.522,E2 21402.522} C_VEL
LIN {X 0,Y 457.059,Z 598.858,A -85,B 0,C 180,E1 21398.841,E2 21398.841} C_VEL
LIN {X 0,Y 457.075,Z 598.858,A -85,B 0,C 180,E1 21395.165,E2 21395.165} C_VEL
LIN {X 0,Y 457.068,Z 598.865,A -85,B 0,C 180,E1 21391.517,E2 21391.517} C_VEL
LIN {X 0,Y 457.045,Z 598.863,A -85,B 0,C 180,E1 21387.846,E2 21387.846} C_VEL
LIN {X 0,Y 457.1,Z 599.076,A -85,B 0,C 180,E1 21384.441,E2 21384.441} C_VEL
LIN {X 0,Y 461.873,Z 614.373,A -85,B 0,C 180,E1 21381.589,E2 21381.589} C_VEL
LIN {X 0,Y 465.449,Z 628.202,A -85,B 0,C 180,E1 21379.228,E2 21379.228} C_VEL
LIN {X 0,Y 463.268,Z 657.122,A -85,B 0,C 180,E1 21375.241,E2 21375.241} C_VEL
LIN {X 0,Y 461.413,Z 685.78,A -85,B 0,C 180,E1 21371.37,E2 21371.37} C_VEL
LIN {X 0,Y 460.211,Z 708.384,A -85,B 0,C 180,E1 21368.387,E2 21368.387} C_VEL
LIN {X 0,Y 463.38,Z 726.826,A -85,B 0,C 180,E1 21367.858,E2 21367.858} C_VEL
LIN {X 0,Y 462.265,Z 808.171,A -85,B 0,C 180,E1 21366.517,E2 21366.517} C_VEL
LIN {X 0,Y 461.22,Z 815.845,A -85,B 0,C 180,E1 21366.439,E2 21366.439} C_VEL
LIN {X 0,Y 455.845,Z 832.885,A -85,B 0,C 180,E1 21366.33,E2 21366.33} C_VEL
LIN {X 0,Y 454.372,Z 840.406,A -85,B 0,C 180,E1 21366.143,E2 21366.143} C_VEL
LIN {X 0,Y 454.236,Z 842.469,A -85,B 0,C 180,E1 21366.065,E2 21366.065} C_VEL
LIN {X 0,Y 453.667,Z 856.854,A -85,B 0,C 180,E1 21365.366,E2 21365.366} C_VEL
LIN {X 0,Y 452.917,Z 871.124,A -85,B 0,C 180,E1 21364.412,E2 21364.412} C_VEL
LIN {X 0,Y 452.042,Z 884.795,A -85,B 0,C 180,E1 21363.191,E2 21363.191} C_VEL
LIN {X 0,Y 451.286,Z 895.643,A -85,B 0,C 180,E1 21361.943,E2 21361.943} C_VEL
LIN {X 0,Y 450.537,Z 905.851,A -85,B 0,C 180,E1 21360.471,E2 21360.471} C_VEL
LIN {X 0,Y 449.861,Z 914.653,A -85,B 0,C 180,E1 21358.836,E2 21358.836} C_VEL
LIN {X 0,Y 449.356,Z 921.751,A -85,B 0,C 180,E1 21357.121,E2 21357.121} C_VEL
LIN {X 0,Y 448.98,Z 927.606,A -85,B 0,C 180,E1 21355.173,E2 21355.173} C_VEL
LIN {X 0,Y 448.763,Z 931.389,A -85,B 0,C 180,E1 21353.226,E2 21353.226} C_VEL
LIN {X 0,Y 448.66,Z 933.358,A -85,B 0,C 180,E1 21351.3,E2 21351.3} C_VEL
LIN {X 0,Y 448.636,Z 933.583,A -85,B 0,C 180,E1 21349.259,E2 21349.259} C_VEL
LIN {X 0,Y 448.688,Z 931.905,A -85,B 0,C 180,E1 21347.24,E2 21347.24} C_VEL
LIN {X 0,Y 448.834,Z 928.656,A -85,B 0,C 180,E1 21345.372,E2 21345.372} C_VEL
LIN {X 0,Y 449.131,Z 923.188,A -85,B 0,C 180,E1 21343.379,E2 21343.379} C_VEL
LIN {X 0,Y 449.572,Z 916.041,A -85,B 0,C 180,E1 21341.546,E2 21341.546} C_VEL
LIN {X 0,Y 450.128,Z 908.028,A -85,B 0,C 180,E1 21339.977,E2 21339.977} C_VEL
LIN {X 0,Y 450.85,Z 897.82,A -85,B 0,C 180,E1 21338.416,E2 21338.416} C_VEL
LIN {X 0,Y 451.571,Z 886.458,A -85,B 0,C 180,E1 21337.059,E2 21337.059} C_VEL
LIN {X 0,Y 452.34,Z 874.186,A -85,B 0,C 180,E1 21335.905,E2 21335.905} C_VEL
LIN {X 0,Y 453.091,Z 860.068,A -85,B 0,C 180,E1 21334.891,E2 21334.891} C_VEL
LIN {X 0,Y 453.676,Z 845.739,A -85,B 0,C 180,E1 21334.139,E2 21334.139} C_VEL
LIN {X 0,Y 454.093,Z 830.685,A -85,B 0,C 180,E1 21333.598,E2 21333.598} C_VEL
LIN {X 0,Y 454.387,Z 809.269,A -85,B 0,C 180,E1 21333.175,E2 21333.175} C_VEL
LIN {X 0,Y 455.275,Z 725.413,A -85,B 0,C 180,E1 21331.786,E2 21331.786} C_VEL
LIN {X 0,Y 452.253,Z 708.568,A -85,B 0,C 180,E1 21331.33,E2 21331.33} C_VEL
LIN {X 0,Y 453.187,Z 689.713,A -85,B 0,C 180,E1 21328.862,E2 21328.862} C_VEL
LIN {X 0,Y 454.974,Z 660.757,A -85,B 0,C 180,E1 21324.957,E2 21324.957} C_VEL
LIN {X 0,Y 456.961,Z 632.29,A -85,B 0,C 180,E1 21321.062,E2 21321.062} C_VEL
LIN {X 0,Y 457.152,Z 628.57,A -85,B 0,C 180,E1 21320.544,E2 21320.544} C_VEL
LIN {X 0,Y 452.38,Z 611.047,A -85,B 0,C 180,E1 21317.62,E2 21317.62} C_VEL
LIN {X 0,Y 449.142,Z 599.976,A -85,B 0,C 180,E1 21315.661,E2 21315.661} C_VEL
LIN {X 0,Y 449.122,Z 599.85,A -85,B 0,C 180,E1 21311.839,E2 21311.839} C_VEL
LIN {X 0,Y 449.133,Z 599.848,A -85,B 0,C 180,E1 21308.037,E2 21308.037} C_VEL
LIN {X 0,Y 449.131,Z 599.841,A -85,B 0,C 180,E1 21304.271,E2 21304.271} C_VEL
LIN {X 0,Y 449.134,Z 599.824,A -85,B 0,C 180,E1 21300.511,E2 21300.511} C_VEL
LIN {X 0,Y 449.12,Z 599.837,A -85,B 0,C 180,E1 21296.793,E2 21296.793} C_VEL
LIN {X 0,Y 449.113,Z 599.848,A -85,B 0,C 180,E1 21293.051,E2 21293.051} C_VEL
LIN {X 0,Y 449.131,Z 599.849,A -85,B 0,C 180,E1 21289.286,E2 21289.286} C_VEL
LIN {X 0,Y 449.135,Z 599.848,A -85,B 0,C 180,E1 21285.472,E2 21285.472} C_VEL
LIN {X 0,Y 449.135,Z 599.835,A -85,B 0,C 180,E1 21281.731,E2 21281.731} C_VEL
LIN {X 0,Y 449.116,Z 599.852,A -85,B 0,C 180,E1 21277.991,E2 21277.991} C_VEL
LIN {X 0,Y 449.106,Z 599.837,A -85,B 0,C 180,E1 21274.282,E2 21274.282} C_VEL
LIN {X 0,Y 449.133,Z 599.848,A -85,B 0,C 180,E1 21270.651,E2 21270.651} C_VEL
LIN {X 0,Y 449.136,Z 599.83,A -85,B 0,C 180,E1 21267.01,E2 21267.01} C_VEL
LIN {X 0,Y 449.113,Z 599.847,A -85,B 0,C 180,E1 21263.346,E2 21263.346} C_VEL
LIN {X 0,Y 449.102,Z 599.847,A -85,B 0,C 180,E1 21259.645,E2 21259.645} C_VEL
LIN {X 0,Y 449.115,Z 599.839,A -85,B 0,C 180,E1 21255.893,E2 21255.893} C_VEL
LIN {X 0,Y 449.137,Z 599.846,A -85,B 0,C 180,E1 21252.21,E2 21252.21} C_VEL
LIN {X 0,Y 449.128,Z 599.828,A -85,B 0,C 180,E1 21248.449,E2 21248.449} C_VEL
LIN {X 0,Y 449.098,Z 599.852,A -85,B 0,C 180,E1 21244.853,E2 21244.853} C_VEL
LIN {X 0,Y 449.1,Z 599.832,A -85,B 0,C 180,E1 21241.148,E2 21241.148} C_VEL
LIN {X 0,Y 449.136,Z 599.849,A -85,B 0,C 180,E1 21237.576,E2 21237.576} C_VEL
LIN {X 0,Y 449.128,Z 599.836,A -85,B 0,C 180,E1 21233.866,E2 21233.866} C_VEL
LIN {X 0,Y 449.091,Z 599.85,A -85,B 0,C 180,E1 21230.259,E2 21230.259} C_VEL
LIN {X 0,Y 449.093,Z 599.843,A -85,B 0,C 180,E1 21226.481,E2 21226.481} C_VEL
LIN {X 0,Y 449.134,Z 599.85,A -85,B 0,C 180,E1 21222.911,E2 21222.911} C_VEL
LIN {X 0,Y 449.137,Z 599.838,A -85,B 0,C 180,E1 21219.134,E2 21219.134} C_VEL
LIN {X 0,Y 449.094,Z 599.856,A -85,B 0,C 180,E1 21215.537,E2 21215.537} C_VEL
LIN {X 0,Y 449.087,Z 599.854,A -85,B 0,C 180,E1 21211.836,E2 21211.836} C_VEL
LIN {X 0,Y 449.128,Z 599.848,A -85,B 0,C 180,E1 21208.258,E2 21208.258} C_VEL
LIN {X 0,Y 449.134,Z 599.845,A -85,B 0,C 180,E1 21204.567,E2 21204.567} C_VEL
LIN {X 0,Y 449.091,Z 599.849,A -85,B 0,C 180,E1 21200.945,E2 21200.945} C_VEL
LIN {X 0,Y 449.085,Z 599.856,A -85,B 0,C 180,E1 21197.23,E2 21197.23} C_VEL
LIN {X 0,Y 449.121,Z 599.85,A -85,B 0,C 180,E1 21193.642,E2 21193.642} C_VEL
LIN {X 0,Y 449.135,Z 599.851,A -85,B 0,C 180,E1 21190.021,E2 21190.021} C_VEL
LIN {X 0,Y 449.115,Z 600.09,A -85,B 0,C 180,E1 21188.958,E2 21188.958} C_VEL
LIN {X 0,Y 456.491,Z 620.663,A -85,B 0,C 180,E1 21186.184,E2 21186.184} C_VEL
LIN {X 0,Y 461.778,Z 636.504,A -85,B 0,C 180,E1 21184.225,E2 21184.225} C_VEL
LIN {X 0,Y 458.315,Z 683.227,A -85,B 0,C 180,E1 21180.045,E2 21180.045} C_VEL
LIN {X 0,Y 457.745,Z 693.627,A -85,B 0,C 180,E1 21179.17,E2 21179.17} C_VEL
LIN {X 0,Y 460.138,Z 714.013,A -85,B 0,C 180,E1 21178.698,E2 21178.698} C_VEL
LIN {X 0,Y 457.839,Z 896.074,A -85,B 0,C 180,E1 21175.807,E2 21175.807} C_VEL
LIN {X 0,Y 457.103,Z 914.969,A -85,B 0,C 180,E1 21175.283,E2 21175.283} C_VEL
LIN {X 0,Y 456.174,Z 932.614,A -85,B 0,C 180,E1 21174.573,E2 21174.573} C_VEL
LIN {X 0,Y 455.104,Z 950.132,A -85,B 0,C 180,E1 21173.631,E2 21173.631} C_VEL
LIN {X 0,Y 453.894,Z 967.139,A -85,B 0,C 180,E1 21172.47,E2 21172.47} C_VEL
LIN {X 0,Y 452.695,Z 983.32,A -85,B 0,C 180,E1 21171.101,E2 21171.101} C_VEL
LIN {X 0,Y 451.502,Z 999.123,A -85,B 0,C 180,E1 21169.469,E2 21169.469} C_VEL
LIN {X 0,Y 450.468,Z 1013.226,A -85,B 0,C 180,E1 21167.703,E2 21167.703} C_VEL
LIN {X 0,Y 449.641,Z 1025.376,A -85,B 0,C 180,E1 21165.874,E2 21165.874} C_VEL
LIN {X 0,Y 449.008,Z 1036.5,A -85,B 0,C 180,E1 21163.859,E2 21163.859} C_VEL
LIN {X 0,Y 448.557,Z 1046.226,A -85,B 0,C 180,E1 21161.704,E2 21161.704} C_VEL
LIN {X 0,Y 448.327,Z 1054.166,A -85,B 0,C 180,E1 21159.5,E2 21159.5} C_VEL
LIN {X 0,Y 448.227,Z 1060.26,A -85,B 0,C 180,E1 21157.305,E2 21157.305} C_VEL
LIN {X 0,Y 448.214,Z 1064.664,A -85,B 0,C 180,E1 21155.12,E2 21155.12} C_VEL
LIN {X 0,Y 448.246,Z 1067.597,A -85,B 0,C 180,E1 21152.813,E2 21152.813} C_VEL
LIN {X 0,Y 448.274,Z 1068.808,A -85,B 0,C 180,E1 21150.511,E2 21150.511} C_VEL
LIN {X 0,Y 448.268,Z 1068.318,A -85,B 0,C 180,E1 21148.211,E2 21148.211} C_VEL
LIN {X 0,Y 448.241,Z 1066.12,A -85,B 0,C 180,E1 21145.907,E2 21145.907} C_VEL
LIN {X 0,Y 448.235,Z 1062.168,A -85,B 0,C 180,E1 21143.597,E2 21143.597} C_VEL
LIN {X 0,Y 448.296,Z 1056.362,A -85,B 0,C 180,E1 21141.277,E2 21141.277} C_VEL
LIN {X 0,Y 448.484,Z 1048.553,A -85,B 0,C 180,E1 21138.946,E2 21138.946} C_VEL
LIN {X 0,Y 448.869,Z 1039.131,A -85,B 0,C 180,E1 21136.736,E2 21136.736} C_VEL
LIN {X 0,Y 449.451,Z 1028.153,A -85,B 0,C 180,E1 21134.649,E2 21134.649} C_VEL
LIN {X 0,Y 450.259,Z 1015.654,A -85,B 0,C 180,E1 21132.689,E2 21132.689} C_VEL
LIN {X 0,Y 451.274,Z 1001.568,A -85,B 0,C 180,E1 21130.858,E2 21130.858} C_VEL
LIN {X 0,Y 452.432,Z 986.046,A -85,B 0,C 180,E1 21129.198,E2 21129.198} C_VEL
LIN {X 0,Y 453.608,Z 969.972,A -85,B 0,C 180,E1 21127.786,E2 21127.786} C_VEL
LIN {X 0,Y 454.798,Z 953.66,A -85,B 0,C 180,E1 21126.62,E2 21126.62} C_VEL
LIN {X 0,Y 455.917,Z 935.965,A -85,B 0,C 180,E1 21125.616,E2 21125.616} C_VEL
LIN {X 0,Y 456.91,Z 917.509,A -85,B 0,C 180,E1 21124.827,E2 21124.827} C_VEL
LIN {X 0,Y 457.717,Z 898.073,A -85,B 0,C 180,E1 21124.255,E2 21124.255} C_VEL
LIN {X 0,Y 458.185,Z 869.501,A -85,B 0,C 180,E1 21123.763,E2 21123.763} C_VEL
LIN {X 0,Y 459.989,Z 711.101,A -85,B 0,C 180,E1 21121.242,E2 21121.242} C_VEL
LIN {X 0,Y 457.776,Z 693.06,A -85,B 0,C 180,E1 21120.78,E2 21120.78} C_VEL
LIN {X 0,Y 460.995,Z 650.501,A -85,B 0,C 180,E1 21116.942,E2 21116.942} C_VEL
LIN {X 0,Y 462.013,Z 636.274,A -85,B 0,C 180,E1 21115.609,E2 21115.609} C_VEL
LIN {X 0,Y 456.05,Z 618.327,A -85,B 0,C 180,E1 21113.235,E2 21113.235} C_VEL
LIN {X 0,Y 450.296,Z 603.251,A -85,B 0,C 180,E1 21111.001,E2 21111.001} C_VEL
LIN {X 0,Y 449.157,Z 600.048,A -85,B 0,C 180,E1 21110.457,E2 21110.457} C_VEL
LIN {X 0,Y 449.083,Z 599.853,A -85,B 0,C 180,E1 21106.881,E2 21106.881} C_VEL
LIN {X 0,Y 449.082,Z 599.86,A -85,B 0,C 180,E1 21103.09,E2 21103.09} C_VEL
LIN {X 0,Y 449.129,Z 599.851,A -85,B 0,C 180,E1 21099.546,E2 21099.546} C_VEL
LIN {X 0,Y 449.13,Z 599.847,A -85,B 0,C 180,E1 21095.838,E2 21095.838} C_VEL
LIN {X 0,Y 449.091,Z 599.85,A -85,B 0,C 180,E1 21092.217,E2 21092.217} C_VEL
LIN {X 0,Y 449.085,Z 599.849,A -85,B 0,C 180,E1 21088.599,E2 21088.599} C_VEL
LIN {X 0,Y 449.129,Z 599.851,A -85,B 0,C 180,E1 21085.023,E2 21085.023} C_VEL
LIN {X 0,Y 449.137,Z 599.85,A -85,B 0,C 180,E1 21081.276,E2 21081.276} C_VEL
LIN {X 0,Y 449.095,Z 599.85,A -85,B 0,C 180,E1 21077.625,E2 21077.625} C_VEL
LIN {X 0,Y 449.087,Z 599.845,A -85,B 0,C 180,E1 21073.898,E2 21073.898} C_VEL
LIN {X 0,Y 449.114,Z 599.841,A -85,B 0,C 180,E1 21070.255,E2 21070.255} C_VEL
LIN {X 0,Y 449.144,Z 599.852,A -85,B 0,C 180,E1 21066.519,E2 21066.519} C_VEL
LIN {X 0,Y 449.114,Z 599.85,A -85,B 0,C 180,E1 21062.807,E2 21062.807} C_VEL
LIN {X 0,Y 449.093,Z 599.846,A -85,B 0,C 180,E1 21059.234,E2 21059.234} C_VEL
LIN {X 0,Y 449.11,Z 599.841,A -85,B 0,C 180,E1 21055.531,E2 21055.531} C_VEL
LIN {X 0,Y 449.139,Z 599.845,A -85,B 0,C 180,E1 21051.809,E2 21051.809} C_VEL
LIN {X 0,Y 449.128,Z 599.852,A -85,B 0,C 180,E1 21048.051,E2 21048.051} C_VEL
LIN {X 0,Y 449.103,Z 599.854,A -85,B 0,C 180,E1 21044.372,E2 21044.372} C_VEL
LIN {X 0,Y 449.104,Z 599.854,A -85,B 0,C 180,E1 21040.626,E2 21040.626} C_VEL
LIN {X 0,Y 449.129,Z 599.848,A -85,B 0,C 180,E1 21036.932,E2 21036.932} C_VEL
LIN {X 0,Y 449.139,Z 599.845,A -85,B 0,C 180,E1 21033.133,E2 21033.133} C_VEL
LIN {X 0,Y 449.135,Z 599.853,A -85,B 0,C 180,E1 21029.349,E2 21029.349} C_VEL
LIN {X 0,Y 449.109,Z 599.853,A -85,B 0,C 180,E1 21025.686,E2 21025.686} C_VEL
LIN {X 0,Y 449.196,Z 600.26,A -85,B 0,C 180,E1 21025.067,E2 21025.067} C_VEL
LIN {X 0,Y 454.126,Z 615.793,A -85,B 0,C 180,E1 21022.1,E2 21022.1} C_VEL
LIN {X 0,Y 458.098,Z 630.509,A -85,B 0,C 180,E1 21019.508,E2 21019.508} C_VEL
LIN {X 0,Y 455.861,Z 658.424,A -85,B 0,C 180,E1 21015.599,E2 21015.599} C_VEL
LIN {X 0,Y 453.853,Z 687.365,A -85,B 0,C 180,E1 21011.631,E2 21011.631} C_VEL
LIN {X 0,Y 452.643,Z 708.001,A -85,B 0,C 180,E1 21008.854,E2 21008.854} C_VEL
LIN {X 0,Y 454.104,Z 716.012,A -85,B 0,C 180,E1 21008.581,E2 21008.581} C_VEL
LIN {X 0,Y 456.09,Z 728.023,A -85,B 0,C 180,E1 21008.255,E2 21008.255} C_VEL
LIN {X 0,Y 454.61,Z 827.537,A -85,B 0,C 180,E1 21006.547,E2 21006.547} C_VEL
LIN {X 0,Y 454.236,Z 842.469,A -85,B 0,C 180,E1 21006.065,E2 21006.065} C_VEL
LIN {X 0,Y 453.077,Z 849.85,A -85,B 0,C 180,E1 21005.793,E2 21005.793} C_VEL
LIN {X 0,Y 447.957,Z 863.963,A -85,B 0,C 180,E1 21005.226,E2 21005.226} C_VEL
LIN {X 0,Y 445.636,Z 871.75,A -85,B 0,C 180,E1 21004.765,E2 21004.765} C_VEL
LIN {X 0,Y 445.256,Z 874.552,A -85,B 0,C 180,E1 21004.546,E2 21004.546} C_VEL
LIN {X 0,Y 444.424,Z 886.624,A -85,B 0,C 180,E1 21003.418,E2 21003.418} C_VEL
LIN {X 0,Y 443.528,Z 898.503,A -85,B 0,C 180,E1 21001.99,E2 21001.99} C_VEL
LIN {X 0,Y 442.751,Z 908.019,A -85,B 0,C 180,E1 21000.538,E2 21000.538} C_VEL
LIN {X 0,Y 442.014,Z 916.937,A -85,B 0,C 180,E1 20998.804,E2 20998.804} C_VEL
LIN {X 0,Y 441.446,Z 924.125,A -85,B 0,C 180,E1 20996.936,E2 20996.936} C_VEL
LIN {X 0,Y 441.081,Z 929.286,A -85,B 0,C 180,E1 20995.081,E2 20995.081} C_VEL
LIN {X 0,Y 440.858,Z 932.89,A -85,B 0,C 180,E1 20993.101,E2 20993.101} C_VEL
LIN {X 0,Y 440.748,Z 934.643,A -85,B 0,C 180,E1 20991.143,E2 20991.143} C_VEL
LIN {X 0,Y 440.726,Z 934.761,A -85,B 0,C 180,E1 20989.205,E2 20989.205} C_VEL
LIN {X 0,Y 440.786,Z 933.036,A -85,B 0,C 180,E1 20987.151,E2 20987.151} C_VEL
LIN {X 0,Y 440.95,Z 929.75,A -85,B 0,C 180,E1 20985.25,E2 20985.25} C_VEL
LIN {X 0,Y 441.278,Z 924.278,A -85,B 0,C 180,E1 20983.229,E2 20983.229} C_VEL
LIN {X 0,Y 441.763,Z 917.08,A -85,B 0,C 180,E1 20981.356,E2 20981.356} C_VEL
LIN {X 0,Y 442.364,Z 909.042,A -85,B 0,C 180,E1 20979.76,E2 20979.76} C_VEL
LIN {X 0,Y 443.137,Z 898.81,A -85,B 0,C 180,E1 20978.172,E2 20978.172} C_VEL
LIN {X 0,Y 443.908,Z 887.431,A -85,B 0,C 180,E1 20976.791,E2 20976.791} C_VEL
LIN {X 0,Y 444.728,Z 875.084,A -85,B 0,C 180,E1 20975.612,E2 20975.612} C_VEL
LIN {X 0,Y 445.531,Z 860.769,A -85,B 0,C 180,E1 20974.569,E2 20974.569} C_VEL
LIN {X 0,Y 446.159,Z 846.068,A -85,B 0,C 180,E1 20973.79,E2 20973.79} C_VEL
LIN {X 0,Y 446.588,Z 831.073,A -85,B 0,C 180,E1 20973.249,E2 20973.249} C_VEL
LIN {X 0,Y 446.901,Z 809.35,A -85,B 0,C 180,E1 20972.816,E2 20972.816} C_VEL
LIN {X 0,Y 447.842,Z 726.435,A -85,B 0,C 180,E1 20971.419,E2 20971.419} C_VEL
LIN {X 0,Y 444.607,Z 708.163,A -85,B 0,C 180,E1 20970.902,E2 20970.902} C_VEL
LIN {X 0,Y 446.315,Z 678.59,A -85,B 0,C 180,E1 20966.918,E2 20966.918} C_VEL
LIN {X 0,Y 448.302,Z 649.952,A -85,B 0,C 180,E1 20962.98,E2 20962.98} C_VEL
LIN {X 0,Y 449.645,Z 630.982,A -85,B 0,C 180,E1 20960.335,E2 20960.335} C_VEL
LIN {X 0,Y 444.72,Z 612.911,A -85,B 0,C 180,E1 20957.271,E2 20957.271} C_VEL
LIN {X 0,Y 441.207,Z 600.957,A -85,B 0,C 180,E1 20955.095,E2 20955.095} C_VEL
LIN {X 0,Y 441.191,Z 600.843,A -85,B 0,C 180,E1 20951.318,E2 20951.318} C_VEL
LIN {X 0,Y 441.178,Z 600.827,A -85,B 0,C 180,E1 20947.619,E2 20947.619} C_VEL
LIN {X 0,Y 441.188,Z 600.837,A -85,B 0,C 180,E1 20943.773,E2 20943.773} C_VEL
LIN {X 0,Y 441.194,Z 600.805,A -85,B 0,C 180,E1 20940.094,E2 20940.094} C_VEL
LIN {X 0,Y 441.194,Z 600.833,A -85,B 0,C 180,E1 20936.273,E2 20936.273} C_VEL
LIN {X 0,Y 441.189,Z 600.831,A -85,B 0,C 180,E1 20932.437,E2 20932.437} C_VEL
LIN {X 0,Y 441.175,Z 600.842,A -85,B 0,C 180,E1 20928.737,E2 20928.737} C_VEL
LIN {X 0,Y 441.184,Z 600.837,A -85,B 0,C 180,E1 20924.999,E2 20924.999} C_VEL
LIN {X 0,Y 441.202,Z 600.817,A -85,B 0,C 180,E1 20921.202,E2 20921.202} C_VEL
LIN {X 0,Y 441.199,Z 600.84,A -85,B 0,C 180,E1 20917.399,E2 20917.399} C_VEL
LIN {X 0,Y 441.19,Z 600.82,A -85,B 0,C 180,E1 20913.572,E2 20913.572} C_VEL
LIN {X 0,Y 441.166,Z 600.842,A -85,B 0,C 180,E1 20909.908,E2 20909.908} C_VEL
LIN {X 0,Y 441.172,Z 600.817,A -85,B 0,C 180,E1 20906.17,E2 20906.17} C_VEL
LIN {X 0,Y 441.198,Z 600.837,A -85,B 0,C 180,E1 20902.379,E2 20902.379} C_VEL
LIN {X 0,Y 441.196,Z 600.817,A -85,B 0,C 180,E1 20898.635,E2 20898.635} C_VEL
LIN {X 0,Y 441.184,Z 600.835,A -85,B 0,C 180,E1 20894.839,E2 20894.839} C_VEL
LIN {X 0,Y 441.161,Z 600.839,A -85,B 0,C 180,E1 20891.108,E2 20891.108} C_VEL
LIN {X 0,Y 441.161,Z 600.827,A -85,B 0,C 180,E1 20887.292,E2 20887.292} C_VEL
LIN {X 0,Y 441.188,Z 600.834,A -85,B 0,C 180,E1 20883.638,E2 20883.638} C_VEL
LIN {X 0,Y 441.203,Z 600.818,A -85,B 0,C 180,E1 20879.87,E2 20879.87} C_VEL
LIN {X 0,Y 441.177,Z 600.846,A -85,B 0,C 180,E1 20876.102,E2 20876.102} C_VEL
LIN {X 0,Y 441.148,Z 600.821,A -85,B 0,C 180,E1 20872.446,E2 20872.446} C_VEL
LIN {X 0,Y 441.167,Z 600.841,A -85,B 0,C 180,E1 20868.761,E2 20868.761} C_VEL
LIN {X 0,Y 441.2,Z 600.825,A -85,B 0,C 180,E1 20865.028,E2 20865.028} C_VEL
LIN {X 0,Y 441.196,Z 600.836,A -85,B 0,C 180,E1 20861.228,E2 20861.228} C_VEL
LIN {X 0,Y 441.152,Z 600.839,A -85,B 0,C 180,E1 20857.619,E2 20857.619} C_VEL
LIN {X 0,Y 441.15,Z 600.83,A -85,B 0,C 180,E1 20853.916,E2 20853.916} C_VEL
LIN {X 0,Y 441.197,Z 600.834,A -85,B 0,C 180,E1 20850.394,E2 20850.394} C_VEL
LIN {X 0,Y 441.2,Z 600.839,A -85,B 0,C 180,E1 20846.586,E2 20846.586} C_VEL
LIN {X 0,Y 441.16,Z 600.847,A -85,B 0,C 180,E1 20842.92,E2 20842.92} C_VEL
LIN {X 0,Y 441.143,Z 600.847,A -85,B 0,C 180,E1 20839.25,E2 20839.25} C_VEL
LIN {X 0,Y 441.183,Z 600.835,A -85,B 0,C 180,E1 20835.731,E2 20835.731} C_VEL
LIN {X 0,Y 441.202,Z 600.842,A -85,B 0,C 180,E1 20831.955,E2 20831.955} C_VEL
LIN {X 0,Y 441.229,Z 601.109,A -85,B 0,C 180,E1 20829.552,E2 20829.552} C_VEL
LIN {X 0,Y 449.115,Z 623.099,A -85,B 0,C 180,E1 20826.516,E2 20826.516} C_VEL
LIN {X 0,Y 454.431,Z 638.907,A -85,B 0,C 180,E1 20824.519,E2 20824.519} C_VEL
LIN {X 0,Y 450.777,Z 685.098,A -85,B 0,C 180,E1 20820.306,E2 20820.306} C_VEL
LIN {X 0,Y 450.254,Z 693.288,A -85,B 0,C 180,E1 20819.592,E2 20819.592} C_VEL
LIN {X 0,Y 452.748,Z 715.075,A -85,B 0,C 180,E1 20819.071,E2 20819.071} C_VEL
LIN {X 0,Y 450.357,Z 895.301,A -85,B 0,C 180,E1 20816.175,E2 20816.175} C_VEL
LIN {X 0,Y 449.586,Z 914.212,A -85,B 0,C 180,E1 20815.644,E2 20815.644} C_VEL
LIN {X 0,Y 448.589,Z 932.043,A -85,B 0,C 180,E1 20814.915,E2 20814.915} C_VEL
LIN {X 0,Y 447.444,Z 949.763,A -85,B 0,C 180,E1 20813.943,E2 20813.943} C_VEL
LIN {X 0,Y 446.151,Z 966.933,A -85,B 0,C 180,E1 20812.743,E2 20812.743} C_VEL
LIN {X 0,Y 444.834,Z 983.679,A -85,B 0,C 180,E1 20811.285,E2 20811.285} C_VEL
LIN {X 0,Y 443.637,Z 998.679,A -85,B 0,C 180,E1 20809.691,E2 20809.691} C_VEL
LIN {X 0,Y 442.555,Z 1012.687,A -85,B 0,C 180,E1 20807.895,E2 20807.895} C_VEL
LIN {X 0,Y 441.641,Z 1025.575,A -85,B 0,C 180,E1 20805.899,E2 20805.899} C_VEL
LIN {X 0,Y 440.985,Z 1036.855,A -85,B 0,C 180,E1 20803.773,E2 20803.773} C_VEL
LIN {X 0,Y 440.546,Z 1046.504,A -85,B 0,C 180,E1 20801.521,E2 20801.521} C_VEL
LIN {X 0,Y 440.343,Z 1054.133,A -85,B 0,C 180,E1 20799.278,E2 20799.278} C_VEL
LIN {X 0,Y 440.27,Z 1059.962,A -85,B 0,C 180,E1 20797.044,E2 20797.044} C_VEL
LIN {X 0,Y 440.285,Z 1064.299,A -85,B 0,C 180,E1 20794.69,E2 20794.69} C_VEL
LIN {X 0,Y 440.335,Z 1066.863,A -85,B 0,C 180,E1 20792.343,E2 20792.343} C_VEL
LIN {X 0,Y 440.367,Z 1067.703,A -85,B 0,C 180,E1 20790,E2 20790} C_VEL
LIN {X 0,Y 440.34,Z 1066.821,A -85,B 0,C 180,E1 20787.658,E2 20787.658} C_VEL
LIN {X 0,Y 440.295,Z 1064.214,A -85,B 0,C 180,E1 20785.311,E2 20785.311} C_VEL
LIN {X 0,Y 440.284,Z 1059.784,A -85,B 0,C 180,E1 20782.932,E2 20782.932} C_VEL
LIN {X 0,Y 440.364,Z 1053.575,A -85,B 0,C 180,E1 20780.591,E2 20780.591} C_VEL
LIN {X 0,Y 440.573,Z 1045.772,A -85,B 0,C 180,E1 20778.347,E2 20778.347} C_VEL
LIN {X 0,Y 441.024,Z 1035.912,A -85,B 0,C 180,E1 20776.095,E2 20776.095} C_VEL
LIN {X 0,Y 441.689,Z 1024.438,A -85,B 0,C 180,E1 20773.968,E2 20773.968} C_VEL
LIN {X 0,Y 442.599,Z 1011.567,A -85,B 0,C 180,E1 20772.001,E2 20772.001} C_VEL
LIN {X 0,Y 443.704,Z 997.127,A -85,B 0,C 180,E1 20770.176,E2 20770.176} C_VEL
LIN {X 0,Y 444.887,Z 982.179,A -85,B 0,C 180,E1 20768.61,E2 20768.61} C_VEL
LIN {X 0,Y 446.189,Z 965.666,A -85,B 0,C 180,E1 20767.19,E2 20767.19} C_VEL
LIN {X 0,Y 447.474,Z 948.512,A -85,B 0,C 180,E1 20766.004,E2 20766.004} C_VEL
LIN {X 0,Y 448.608,Z 931.033,A -85,B 0,C 180,E1 20765.052,E2 20765.052} C_VEL
LIN {X 0,Y 449.644,Z 912.693,A -85,B 0,C 180,E1 20764.308,E2 20764.308} C_VEL
LIN {X 0,Y 450.419,Z 893.558,A -85,B 0,C 180,E1 20763.785,E2 20763.785} C_VEL
LIN {X 0,Y 452.704,Z 712.121,A -85,B 0,C 180,E1 20760.838,E2 20760.838} C_VEL
LIN {X 0,Y 450.414,Z 693.257,A -85,B 0,C 180,E1 20760.347,E2 20760.347} C_VEL
LIN {X 0,Y 453.908,Z 650.803,A -85,B 0,C 180,E1 20756.434,E2 20756.434} C_VEL
LIN {X 0,Y 454.807,Z 639.075,A -85,B 0,C 180,E1 20755.307,E2 20755.307} C_VEL
LIN {X 0,Y 448.713,Z 620.733,A -85,B 0,C 180,E1 20752.808,E2 20752.808} C_VEL
LIN {X 0,Y 443.294,Z 606.756,A -85,B 0,C 180,E1 20750.669,E2 20750.669} C_VEL
LIN {X 0,Y 441.19,Z 601.031,A -85,B 0,C 180,E1 20749.694,E2 20749.694} C_VEL
LIN {X 0,Y 441.198,Z 600.836,A -85,B 0,C 180,E1 20746.095,E2 20746.095} C_VEL
LIN {X 0,Y 441.167,Z 600.845,A -85,B 0,C 180,E1 20742.367,E2 20742.367} C_VEL
LIN {X 0,Y 441.139,Z 600.837,A -85,B 0,C 180,E1 20738.768,E2 20738.768} C_VEL
LIN {X 0,Y 441.161,Z 600.836,A -85,B 0,C 180,E1 20735.097,E2 20735.097} C_VEL
LIN {X 0,Y 441.204,Z 600.829,A -85,B 0,C 180,E1 20731.414,E2 20731.414} C_VEL
LIN {X 0,Y 441.18,Z 600.829,A -85,B 0,C 180,E1 20727.684,E2 20727.684} C_VEL
LIN {X 0,Y 441.149,Z 600.835,A -85,B 0,C 180,E1 20724.021,E2 20724.021} C_VEL
LIN {X 0,Y 441.149,Z 600.838,A -85,B 0,C 180,E1 20720.228,E2 20720.228} C_VEL
LIN {X 0,Y 441.177,Z 600.844,A -85,B 0,C 180,E1 20716.531,E2 20716.531} C_VEL
LIN {X 0,Y 441.198,Z 600.834,A -85,B 0,C 180,E1 20712.832,E2 20712.832} C_VEL
LIN {X 0,Y 441.168,Z 600.825,A -85,B 0,C 180,E1 20709.128,E2 20709.128} C_VEL
LIN {X 0,Y 441.151,Z 600.834,A -85,B 0,C 180,E1 20705.462,E2 20705.462} C_VEL
LIN {X 0,Y 441.163,Z 600.842,A -85,B 0,C 180,E1 20701.688,E2 20701.688} C_VEL
LIN {X 0,Y 441.195,Z 600.838,A -85,B 0,C 180,E1 20698.044,E2 20698.044} C_VEL
LIN {X 0,Y 441.193,Z 600.829,A -85,B 0,C 180,E1 20694.206,E2 20694.206} C_VEL
LIN {X 0,Y 441.161,Z 600.828,A -85,B 0,C 180,E1 20690.608,E2 20690.608} C_VEL
LIN {X 0,Y 441.161,Z 600.831,A -85,B 0,C 180,E1 20686.9,E2 20686.9} C_VEL
LIN {X 0,Y 441.192,Z 600.832,A -85,B 0,C 180,E1 20683.272,E2 20683.272} C_VEL
LIN {X 0,Y 441.2,Z 600.832,A -85,B 0,C 180,E1 20679.435,E2 20679.435} C_VEL
LIN {X 0,Y 441.178,Z 600.832,A -85,B 0,C 180,E1 20675.782,E2 20675.782} C_VEL
LIN {X 0,Y 441.167,Z 600.845,A -85,B 0,C 180,E1 20672.021,E2 20672.021} C_VEL
LIN {X 0,Y 441.176,Z 600.838,A -85,B 0,C 180,E1 20668.278,E2 20668.278} C_VEL
LIN {X 0,Y 441.208,Z 601.114,A -85,B 0,C 180,E1 20665.819,E2 20665.819} C_VEL
LIN {X 0,Y 446.201,Z 616.486,A -85,B 0,C 180,E1 20662.769,E2 20662.769} C_VEL
LIN {X 0,Y 450.423,Z 631.864,A -85,B 0,C 180,E1 20659.982,E2 20659.982} C_VEL
LIN {X 0,Y 450.659,Z 634.548,A -85,B 0,C 180,E1 20659.552,E2 20659.552} C_VEL
LIN {X 0,Y 448.244,Z 662.837,A -85,B 0,C 180,E1 20655.539,E2 20655.539} C_VEL
LIN {X 0,Y 446.137,Z 691.638,A -85,B 0,C 180,E1 20651.535,E2 20651.535} C_VEL
LIN {X 0,Y 445.15,Z 708.189,A -85,B 0,C 180,E1 20649.302,E2 20649.302} C_VEL
LIN {X 0,Y 448.829,Z 728.844,A -85,B 0,C 180,E1 20648.673,E2 20648.673} C_VEL
LIN {X 0,Y 447.24,Z 828.28,A -85,B 0,C 180,E1 20646.932,E2 20646.932} C_VEL
LIN {X 0,Y 446.809,Z 844.392,A -85,B 0,C 180,E1 20646.395,E2 20646.395} C_VEL
LIN {X 0,Y 446.156,Z 859.183,A -85,B 0,C 180,E1 20645.639,E2 20645.639} C_VEL
LIN {X 0,Y 445.372,Z 872.83,A -85,B 0,C 180,E1 20644.688,E2 20644.688} C_VEL
LIN {X 0,Y 445.256,Z 874.552,A -85,B 0,C 180,E1 20644.546,E2 20644.546} C_VEL
LIN {X 0,Y 443.897,Z 881.059,A -85,B 0,C 180,E1 20644.026,E2 20644.026} C_VEL
LIN {X 0,Y 438.51,Z 893.31,A -85,B 0,C 180,E1 20642.972,E2 20642.972} C_VEL
LIN {X 0,Y 436.09,Z 899.779,A -85,B 0,C 180,E1 20642.24,E2 20642.24} C_VEL
LIN {X 0,Y 435.692,Z 902.037,A -85,B 0,C 180,E1 20641.926,E2 20641.926} C_VEL
LIN {X 0,Y 434.859,Z 911.429,A -85,B 0,C 180,E1 20640.387,E2 20640.387} C_VEL
LIN {X 0,Y 434.102,Z 919.751,A -85,B 0,C 180,E1 20638.625,E2 20638.625} C_VEL
LIN {X 0,Y 433.557,Z 926.265,A -85,B 0,C 180,E1 20636.811,E2 20636.811} C_VEL
LIN {X 0,Y 433.145,Z 931.603,A -85,B 0,C 180,E1 20634.697,E2 20634.697} C_VEL
LIN {X 0,Y 432.923,Z 934.682,A -85,B 0,C 180,E1 20632.687,E2 20632.687} C_VEL
LIN {X 0,Y 432.829,Z 936.043,A -85,B 0,C 180,E1 20630.678,E2 20630.678} C_VEL
LIN {X 0,Y 432.829,Z 935.55,A -85,B 0,C 180,E1 20628.45,E2 20628.45} C_VEL
LIN {X 0,Y 432.935,Z 933.155,A -85,B 0,C 180,E1 20626.365,E2 20626.365} C_VEL
LIN {X 0,Y 433.162,Z 929.22,A -85,B 0,C 180,E1 20624.436,E2 20624.436} C_VEL
LIN {X 0,Y 433.589,Z 922.979,A -85,B 0,C 180,E1 20622.384,E2 20622.384} C_VEL
LIN {X 0,Y 434.146,Z 915.586,A -85,B 0,C 180,E1 20620.617,E2 20620.617} C_VEL
LIN {X 0,Y 434.852,Z 906.866,A -85,B 0,C 180,E1 20618.995,E2 20618.995} C_VEL
LIN {X 0,Y 435.725,Z 895.716,A -85,B 0,C 180,E1 20617.383,E2 20617.383} C_VEL
LIN {X 0,Y 436.56,Z 883.885,A -85,B 0,C 180,E1 20616.047,E2 20616.047} C_VEL
LIN {X 0,Y 437.432,Z 871.095,A -85,B 0,C 180,E1 20614.917,E2 20614.917} C_VEL
LIN {X 0,Y 438.239,Z 856.187,A -85,B 0,C 180,E1 20613.925,E2 20613.925} C_VEL
LIN {X 0,Y 438.826,Z 841.18,A -85,B 0,C 180,E1 20613.216,E2 20613.216} C_VEL
LIN {X 0,Y 439.195,Z 825.901,A -85,B 0,C 180,E1 20612.748,E2 20612.748} C_VEL
LIN {X 0,Y 440.43,Z 727.484,A -85,B 0,C 180,E1 20611.04,E2 20611.04} C_VEL
LIN {X 0,Y 436.995,Z 708.152,A -85,B 0,C 180,E1 20610.491,E2 20610.491} C_VEL
LIN {X 0,Y 438.739,Z 679.664,A -85,B 0,C 180,E1 20606.603,E2 20606.603} C_VEL
LIN {X 0,Y 440.786,Z 651.647,A -85,B 0,C 180,E1 20602.702,E2 20602.702} C_VEL
LIN {X 0,Y 442.116,Z 633.302,A -85,B 0,C 180,E1 20600.103,E2 20600.103} C_VEL
LIN {X 0,Y 437.183,Z 615.18,A -85,B 0,C 180,E1 20596.979,E2 20596.979} C_VEL
LIN {X 0,Y 433.272,Z 601.947,A -85,B 0,C 180,E1 20594.541,E2 20594.541} C_VEL
LIN {X 0,Y 433.254,Z 601.827,A -85,B 0,C 180,E1 20590.716,E2 20590.716} C_VEL
LIN {X 0,Y 433.256,Z 601.796,A -85,B 0,C 180,E1 20586.9,E2 20586.9} C_VEL
LIN {X 0,Y 433.246,Z 601.83,A -85,B 0,C 180,E1 20583.106,E2 20583.106} C_VEL
LIN {X 0,Y 433.234,Z 601.786,A -85,B 0,C 180,E1 20579.333,E2 20579.333} C_VEL
LIN {X 0,Y 433.249,Z 601.827,A -85,B 0,C 180,E1 20575.477,E2 20575.477} C_VEL
LIN {X 0,Y 433.261,Z 601.822,A -85,B 0,C 180,E1 20571.626,E2 20571.626} C_VEL
LIN {X 0,Y 433.256,Z 601.814,A -85,B 0,C 180,E1 20567.8,E2 20567.8} C_VEL
LIN {X 0,Y 433.255,Z 601.832,A -85,B 0,C 180,E1 20563.942,E2 20563.942} C_VEL
LIN {X 0,Y 433.235,Z 601.81,A -85,B 0,C 180,E1 20560.189,E2 20560.189} C_VEL
LIN {X 0,Y 433.232,Z 601.829,A -85,B 0,C 180,E1 20556.345,E2 20556.345} C_VEL
LIN {X 0,Y 433.24,Z 601.816,A -85,B 0,C 180,E1 20552.53,E2 20552.53} C_VEL
LIN {X 0,Y 433.262,Z 601.823,A -85,B 0,C 180,E1 20548.837,E2 20548.837} C_VEL
LIN {X 0,Y 433.257,Z 601.808,A -85,B 0,C 180,E1 20544.982,E2 20544.982} C_VEL
LIN {X 0,Y 433.242,Z 601.834,A -85,B 0,C 180,E1 20541.191,E2 20541.191} C_VEL
LIN {X 0,Y 433.22,Z 601.804,A -85,B 0,C 180,E1 20537.46,E2 20537.46} C_VEL
LIN {X 0,Y 433.232,Z 601.828,A -85,B 0,C 180,E1 20533.678,E2 20533.678} C_VEL
LIN {X 0,Y 433.252,Z 601.805,A -85,B 0,C 180,E1 20529.968,E2 20529.968} C_VEL
LIN {X 0,Y 433.262,Z 601.823,A -85,B 0,C 180,E1 20526.227,E2 20526.227} C_VEL
LIN {X 0,Y 433.228,Z 601.821,A -85,B 0,C 180,E1 20522.514,E2 20522.514} C_VEL
LIN {X 0,Y 433.216,Z 601.819,A -85,B 0,C 180,E1 20518.81,E2 20518.81} C_VEL
LIN {X 0,Y 433.235,Z 601.824,A -85,B 0,C 180,E1 20515.102,E2 20515.102} C_VEL
LIN {X 0,Y 433.26,Z 601.816,A -85,B 0,C 180,E1 20511.373,E2 20511.373} C_VEL
LIN {X 0,Y 433.249,Z 601.825,A -85,B 0,C 180,E1 20507.607,E2 20507.607} C_VEL
LIN {X 0,Y 433.211,Z 601.824,A -85,B 0,C 180,E1 20504.059,E2 20504.059} C_VEL
LIN {X 0,Y 433.22,Z 601.823,A -85,B 0,C 180,E1 20500.308,E2 20500.308} C_VEL
LIN {X 0,Y 433.252,Z 601.828,A -85,B 0,C 180,E1 20496.613,E2 20496.613} C_VEL
LIN {X 0,Y 433.262,Z 601.821,A -85,B 0,C 180,E1 20492.811,E2 20492.811} C_VEL
LIN {X 0,Y 433.221,Z 601.823,A -85,B 0,C 180,E1 20489.157,E2 20489.157} C_VEL
LIN {X 0,Y 433.205,Z 601.829,A -85,B 0,C 180,E1 20485.485,E2 20485.485} C_VEL
LIN {X 0,Y 433.227,Z 601.824,A -85,B 0,C 180,E1 20481.792,E2 20481.792} C_VEL
LIN {X 0,Y 433.263,Z 601.823,A -85,B 0,C 180,E1 20478.169,E2 20478.169} C_VEL
LIN {X 0,Y 433.236,Z 601.833,A -85,B 0,C 180,E1 20474.371,E2 20474.371} C_VEL
LIN {X 0,Y 433.202,Z 601.831,A -85,B 0,C 180,E1 20470.783,E2 20470.783} C_VEL
LIN {X 0,Y 433.31,Z 602.26,A -85,B 0,C 180,E1 20470.127,E2 20470.127} C_VEL
LIN {X 0,Y 441.512,Z 624.973,A -85,B 0,C 180,E1 20466.926,E2 20466.926} C_VEL
LIN {X 0,Y 447.053,Z 641.729,A -85,B 0,C 180,E1 20464.773,E2 20464.773} C_VEL
LIN {X 0,Y 443.129,Z 688.533,A -85,B 0,C 180,E1 20460.435,E2 20460.435} C_VEL
LIN {X 0,Y 442.835,Z 693.872,A -85,B 0,C 180,E1 20459.985,E2 20459.985} C_VEL
LIN {X 0,Y 445.363,Z 716.082,A -85,B 0,C 180,E1 20459.454,E2 20459.454} C_VEL
LIN {X 0,Y 442.852,Z 894.874,A -85,B 0,C 180,E1 20456.536,E2 20456.536} C_VEL
LIN {X 0,Y 442.048,Z 913.691,A -85,B 0,C 180,E1 20456,E2 20456} C_VEL
LIN {X 0,Y 440.967,Z 932.068,A -85,B 0,C 180,E1 20455.232,E2 20455.232} C_VEL
LIN {X 0,Y 439.76,Z 949.783,A -85,B 0,C 180,E1 20454.237,E2 20454.237} C_VEL
LIN {X 0,Y 438.417,Z 966.725,A -85,B 0,C 180,E1 20453.025,E2 20453.025} C_VEL
LIN {X 0,Y 437.084,Z 982.646,A -85,B 0,C 180,E1 20451.611,E2 20451.611} C_VEL
LIN {X 0,Y 435.823,Z 997.655,A -85,B 0,C 180,E1 20449.989,E2 20449.989} C_VEL
LIN {X 0,Y 434.71,Z 1011.318,A -85,B 0,C 180,E1 20448.209,E2 20448.209} C_VEL
LIN {X 0,Y 433.746,Z 1024.143,A -85,B 0,C 180,E1 20446.196,E2 20446.196} C_VEL
LIN {X 0,Y 433.049,Z 1035.497,A -85,B 0,C 180,E1 20444.031,E2 20444.031} C_VEL
LIN {X 0,Y 432.587,Z 1045.208,A -85,B 0,C 180,E1 20441.736,E2 20441.736} C_VEL
LIN {X 0,Y 432.383,Z 1052.882,A -85,B 0,C 180,E1 20439.45,E2 20439.45} C_VEL
LIN {X 0,Y 432.321,Z 1058.75,A -85,B 0,C 180,E1 20437.171,E2 20437.171} C_VEL
LIN {X 0,Y 432.351,Z 1063.1,A -85,B 0,C 180,E1 20434.776,E2 20434.776} C_VEL
LIN {X 0,Y 432.417,Z 1065.672,A -85,B 0,C 180,E1 20432.386,E2 20432.386} C_VEL
LIN {X 0,Y 432.457,Z 1066.511,A -85,B 0,C 180,E1 20430,E2 20430} C_VEL
LIN {X 0,Y 432.423,Z 1065.621,A -85,B 0,C 180,E1 20427.615,E2 20427.615} C_VEL
LIN {X 0,Y 432.364,Z 1062.999,A -85,B 0,C 180,E1 20425.225,E2 20425.225} C_VEL
LIN {X 0,Y 432.337,Z 1058.567,A -85,B 0,C 180,E1 20422.811,E2 20422.811} C_VEL
LIN {X 0,Y 432.403,Z 1052.308,A -85,B 0,C 180,E1 20420.417,E2 20420.417} C_VEL
LIN {X 0,Y 432.616,Z 1044.474,A -85,B 0,C 180,E1 20418.13,E2 20418.13} C_VEL
LIN {X 0,Y 433.088,Z 1034.561,A -85,B 0,C 180,E1 20415.835,E2 20415.835} C_VEL
LIN {X 0,Y 433.742,Z 1023.844,A -85,B 0,C 180,E1 20413.804,E2 20413.804} C_VEL
LIN {X 0,Y 434.695,Z 1011.035,A -85,B 0,C 180,E1 20411.797,E2 20411.797} C_VEL
LIN {X 0,Y 435.803,Z 997.311,A -85,B 0,C 180,E1 20410.011,E2 20410.011} C_VEL
LIN {X 0,Y 437.097,Z 981.868,A -85,B 0,C 180,E1 20408.343,E2 20408.343} C_VEL
LIN {X 0,Y 438.506,Z 965.195,A -85,B 0,C 180,E1 20406.871,E2 20406.871} C_VEL
LIN {X 0,Y 439.822,Z 948.781,A -85,B 0,C 180,E1 20405.703,E2 20405.703} C_VEL
LIN {X 0,Y 441.06,Z 930.956,A -85,B 0,C 180,E1 20404.703,E2 20404.703} C_VEL
LIN {X 0,Y 442.15,Z 912.849,A -85,B 0,C 180,E1 20403.947,E2 20403.947} C_VEL
LIN {X 0,Y 442.973,Z 894.074,A -85,B 0,C 180,E1 20403.413,E2 20403.413} C_VEL
LIN {X 0,Y 445.448,Z 713.163,A -85,B 0,C 180,E1 20400.421,E2 20400.421} C_VEL
LIN {X 0,Y 443.092,Z 693.541,A -85,B 0,C 180,E1 20399.9,E2 20399.9} C_VEL
LIN {X 0,Y 446.905,Z 650.776,A -85,B 0,C 180,E1 20395.873,E2 20395.873} C_VEL
LIN {X 0,Y 447.721,Z 642.256,A -85,B 0,C 180,E1 20395.044,E2 20395.044} C_VEL
LIN {X 0,Y 441.906,Z 624.554,A -85,B 0,C 180,E1 20392.577,E2 20392.577} C_VEL
LIN {X 0,Y 435.706,Z 608.3,A -85,B 0,C 180,E1 20390.018,E2 20390.018} C_VEL
LIN {X 0,Y 433.234,Z 602.022,A -85,B 0,C 180,E1 20388.893,E2 20388.893} C_VEL
LIN {X 0,Y 433.203,Z 601.837,A -85,B 0,C 180,E1 20385.119,E2 20385.119} C_VEL
LIN {X 0,Y 433.232,Z 601.826,A -85,B 0,C 180,E1 20381.481,E2 20381.481} C_VEL
LIN {X 0,Y 433.259,Z 601.82,A -85,B 0,C 180,E1 20377.869,E2 20377.869} C_VEL
LIN {X 0,Y 433.223,Z 601.83,A -85,B 0,C 180,E1 20374.113,E2 20374.113} C_VEL
LIN {X 0,Y 433.205,Z 601.834,A -85,B 0,C 180,E1 20370.515,E2 20370.515} C_VEL
LIN {X 0,Y 433.232,Z 601.824,A -85,B 0,C 180,E1 20366.894,E2 20366.894} C_VEL
LIN {X 0,Y 433.264,Z 601.814,A -85,B 0,C 180,E1 20363.098,E2 20363.098} C_VEL
LIN {X 0,Y 433.247,Z 601.816,A -85,B 0,C 180,E1 20359.282,E2 20359.282} C_VEL
LIN {X 0,Y 433.214,Z 601.829,A -85,B 0,C 180,E1 20355.666,E2 20355.666} C_VEL
LIN {X 0,Y 433.212,Z 601.834,A -85,B 0,C 180,E1 20351.853,E2 20351.853} C_VEL
LIN {X 0,Y 433.231,Z 601.826,A -85,B 0,C 180,E1 20348.093,E2 20348.093} C_VEL
LIN {X 0,Y 433.255,Z 601.813,A -85,B 0,C 180,E1 20344.367,E2 20344.367} C_VEL
LIN {X 0,Y 433.253,Z 601.819,A -85,B 0,C 180,E1 20340.529,E2 20340.529} C_VEL
LIN {X 0,Y 433.224,Z 601.83,A -85,B 0,C 180,E1 20336.824,E2 20336.824} C_VEL
LIN {X 0,Y 433.221,Z 601.833,A -85,B 0,C 180,E1 20333.107,E2 20333.107} C_VEL
LIN {X 0,Y 433.241,Z 601.827,A -85,B 0,C 180,E1 20329.36,E2 20329.36} C_VEL
LIN {X 0,Y 433.264,Z 601.82,A -85,B 0,C 180,E1 20325.567,E2 20325.567} C_VEL
LIN {X 0,Y 433.257,Z 601.823,A -85,B 0,C 180,E1 20321.708,E2 20321.708} C_VEL
LIN {X 0,Y 433.238,Z 601.83,A -85,B 0,C 180,E1 20317.902,E2 20317.902} C_VEL
LIN {X 0,Y 433.228,Z 601.832,A -85,B 0,C 180,E1 20314.138,E2 20314.138} C_VEL
LIN {X 0,Y 433.238,Z 601.826,A -85,B 0,C 180,E1 20310.403,E2 20310.403} C_VEL
LIN {X 0,Y 433.283,Z 601.998,A -85,B 0,C 180,E1 20306.615,E2 20306.615} C_VEL
LIN {X 0,Y 438.296,Z 617.3,A -85,B 0,C 180,E1 20303.458,E2 20303.458} C_VEL
LIN {X 0,Y 442.363,Z 631.799,A -85,B 0,C 180,E1 20300.737,E2 20300.737} C_VEL
LIN {X 0,Y 443.38,Z 636.846,A -85,B 0,C 180,E1 20299.86,E2 20299.86} C_VEL
LIN {X 0,Y 440.807,Z 665.125,A -85,B 0,C 180,E1 20295.788,E2 20295.788} C_VEL
LIN {X 0,Y 438.567,Z 693.82,A -85,B 0,C 180,E1 20291.737,E2 20291.737} C_VEL
LIN {X 0,Y 437.656,Z 707.884,A -85,B 0,C 180,E1 20289.804,E2 20289.804} C_VEL
LIN {X 0,Y 439.539,Z 717.88,A -85,B 0,C 180,E1 20289.452,E2 20289.452} C_VEL
LIN {X 0,Y 441.588,Z 730.323,A -85,B 0,C 180,E1 20289.094,E2 20289.094} C_VEL
LIN {X 0,Y 439.894,Z 828.917,A -85,B 0,C 180,E1 20287.333,E2 20287.333} C_VEL
LIN {X 0,Y 439.43,Z 845.2,A -85,B 0,C 180,E1 20286.781,E2 20286.781} C_VEL
LIN {X 0,Y 438.722,Z 860.261,A -85,B 0,C 180,E1 20285.996,E2 20285.996} C_VEL
LIN {X 0,Y 437.889,Z 873.837,A -85,B 0,C 180,E1 20285.031,E2 20285.031} C_VEL
LIN {X 0,Y 436.911,Z 887.194,A -85,B 0,C 180,E1 20283.786,E2 20283.786} C_VEL
LIN {X 0,Y 435.966,Z 898.776,A -85,B 0,C 180,E1 20282.387,E2 20282.387} C_VEL
LIN {X 0,Y 435.692,Z 902.037,A -85,B 0,C 180,E1 20281.926,E2 20281.926} C_VEL
LIN {X 0,Y 434.28,Z 907.216,A -85,B 0,C 180,E1 20281.181,E2 20281.181} C_VEL
LIN {X 0,Y 428.847,Z 916.677,A -85,B 0,C 180,E1 20279.691,E2 20279.691} C_VEL
LIN {X 0,Y 426.496,Z 921.35,A -85,B 0,C 180,E1 20278.729,E2 20278.729} C_VEL
LIN {X 0,Y 426.152,Z 922.892,A -85,B 0,C 180,E1 20278.336,E2 20278.336} C_VEL
LIN {X 0,Y 425.581,Z 929.233,A -85,B 0,C 180,E1 20276.362,E2 20276.362} C_VEL
LIN {X 0,Y 425.197,Z 933.744,A -85,B 0,C 180,E1 20274.3,E2 20274.3} C_VEL
LIN {X 0,Y 424.994,Z 936.39,A -85,B 0,C 180,E1 20272.258,E2 20272.258} C_VEL
LIN {X 0,Y 424.908,Z 937.308,A -85,B 0,C 180,E1 20270.093,E2 20270.093} C_VEL
LIN {X 0,Y 424.931,Z 936.342,A -85,B 0,C 180,E1 20267.953,E2 20267.953} C_VEL
LIN {X 0,Y 425.067,Z 933.813,A -85,B 0,C 180,E1 20265.974,E2 20265.974} C_VEL
LIN {X 0,Y 425.363,Z 929.183,A -85,B 0,C 180,E1 20263.872,E2 20263.872} C_VEL
LIN {X 0,Y 425.79,Z 923.478,A -85,B 0,C 180,E1 20262.063,E2 20262.063} C_VEL
LIN {X 0,Y 426.471,Z 915.271,A -85,B 0,C 180,E1 20260.127,E2 20260.127} C_VEL
LIN {X 0,Y 427.247,Z 906.113,A -85,B 0,C 180,E1 20258.478,E2 20258.478} C_VEL
LIN {X 0,Y 428.123,Z 895.58,A -85,B 0,C 180,E1 20256.975,E2 20256.975} C_VEL
LIN {X 0,Y 429.086,Z 882.783,A -85,B 0,C 180,E1 20255.549,E2 20255.549} C_VEL
LIN {X 0,Y 430.006,Z 869.328,A -85,B 0,C 180,E1 20254.401,E2 20254.401} C_VEL
LIN {X 0,Y 430.759,Z 855.963,A -85,B 0,C 180,E1 20253.527,E2 20253.527} C_VEL
LIN {X 0,Y 431.403,Z 839.96,A -85,B 0,C 180,E1 20252.784,E2 20252.784} C_VEL
LIN {X 0,Y 431.752,Z 824.157,A -85,B 0,C 180,E1 20252.331,E2 20252.331} C_VEL
LIN {X 0,Y 433.062,Z 728.685,A -85,B 0,C 180,E1 20250.653,E2 20250.653} C_VEL
LIN {X 0,Y 429.379,Z 707.712,A -85,B 0,C 180,E1 20250.033,E2 20250.033} C_VEL
LIN {X 0,Y 431.379,Z 677.854,A -85,B 0,C 180,E1 20245.879,E2 20245.879} C_VEL
LIN {X 0,Y 433.564,Z 649.809,A -85,B 0,C 180,E1 20241.913,E2 20241.913} C_VEL
LIN {X 0,Y 434.662,Z 635.914,A -85,B 0,C 180,E1 20239.912,E2 20239.912} C_VEL
LIN {X 0,Y 429.675,Z 617.484,A -85,B 0,C 180,E1 20236.681,E2 20236.681} C_VEL
LIN {X 0,Y 425.321,Z 602.93,A -85,B 0,C 180,E1 20233.952,E2 20233.952} C_VEL
LIN {X 0,Y 425.312,Z 602.812,A -85,B 0,C 180,E1 20230.069,E2 20230.069} C_VEL
LIN {X 0,Y 425.312,Z 602.779,A -85,B 0,C 180,E1 20226.296,E2 20226.296} C_VEL
LIN {X 0,Y 425.318,Z 602.817,A -85,B 0,C 180,E1 20222.409,E2 20222.409} C_VEL
LIN {X 0,Y 425.313,Z 602.772,A -85,B 0,C 180,E1 20218.54,E2 20218.54} C_VEL
LIN {X 0,Y 425.307,Z 602.822,A -85,B 0,C 180,E1 20214.664,E2 20214.664} C_VEL
LIN {X 0,Y 425.299,Z 602.816,A -85,B 0,C 180,E1 20210.771,E2 20210.771} C_VEL
LIN {X 0,Y 425.3,Z 602.8,A -85,B 0,C 180,E1 20206.983,E2 20206.983} C_VEL
LIN {X 0,Y 425.315,Z 602.813,A -85,B 0,C 180,E1 20203.166,E2 20203.166} C_VEL
LIN {X 0,Y 425.321,Z 602.81,A -85,B 0,C 180,E1 20199.337,E2 20199.337} C_VEL
LIN {X 0,Y 425.316,Z 602.806,A -85,B 0,C 180,E1 20195.498,E2 20195.498} C_VEL
LIN {X 0,Y 425.302,Z 602.81,A -85,B 0,C 180,E1 20191.674,E2 20191.674} C_VEL
LIN {X 0,Y 425.29,Z 602.814,A -85,B 0,C 180,E1 20187.873,E2 20187.873} C_VEL
LIN {X 0,Y 425.29,Z 602.808,A -85,B 0,C 180,E1 20184,E2 20184} C_VEL
LIN {X 0,Y 425.311,Z 602.81,A -85,B 0,C 180,E1 20180.218,E2 20180.218} C_VEL
LIN {X 0,Y 425.32,Z 602.797,A -85,B 0,C 180,E1 20176.386,E2 20176.386} C_VEL
LIN {X 0,Y 425.314,Z 602.818,A -85,B 0,C 180,E1 20172.629,E2 20172.629} C_VEL
LIN {X 0,Y 425.283,Z 602.792,A -85,B 0,C 180,E1 20168.927,E2 20168.927} C_VEL
LIN {X 0,Y 425.283,Z 602.817,A -85,B 0,C 180,E1 20165.126,E2 20165.126} C_VEL
LIN {X 0,Y 425.295,Z 602.795,A -85,B 0,C 180,E1 20161.347,E2 20161.347} C_VEL
LIN {X 0,Y 425.319,Z 602.816,A -85,B 0,C 180,E1 20157.575,E2 20157.575} C_VEL
LIN {X 0,Y 425.322,Z 602.795,A -85,B 0,C 180,E1 20153.657,E2 20153.657} C_VEL
LIN {X 0,Y 425.298,Z 602.818,A -85,B 0,C 180,E1 20149.845,E2 20149.845} C_VEL
LIN {X 0,Y 425.271,Z 602.807,A -85,B 0,C 180,E1 20146.125,E2 20146.125} C_VEL
LIN {X 0,Y 425.28,Z 602.82,A -85,B 0,C 180,E1 20142.345,E2 20142.345} C_VEL
LIN {X 0,Y 425.304,Z 602.807,A -85,B 0,C 180,E1 20138.588,E2 20138.588} C_VEL
LIN {X 0,Y 425.321,Z 602.806,A -85,B 0,C 180,E1 20134.818,E2 20134.818} C_VEL
LIN {X 0,Y 425.308,Z 602.821,A -85,B 0,C 180,E1 20130.991,E2 20130.991} C_VEL
LIN {X 0,Y 425.273,Z 602.822,A -85,B 0,C 180,E1 20127.265,E2 20127.265} C_VEL
LIN {X 0,Y 425.27,Z 602.823,A -85,B 0,C 180,E1 20123.5,E2 20123.5} C_VEL
LIN {X 0,Y 425.305,Z 602.821,A -85,B 0,C 180,E1 20119.823,E2 20119.823} C_VEL
LIN {X 0,Y 425.32,Z 602.812,A -85,B 0,C 180,E1 20116.002,E2 20116.002} C_VEL
LIN {X 0,Y 425.303,Z 602.818,A -85,B 0,C 180,E1 20112.222,E2 20112.222} C_VEL
LIN {X 0,Y 425.307,Z 603.12,A -85,B 0,C 180,E1 20110.8,E2 20110.8} C_VEL
LIN {X 0,Y 432.882,Z 624.06,A -85,B 0,C 180,E1 20107.741,E2 20107.741} C_VEL
LIN {X 0,Y 439.695,Z 644.169,A -85,B 0,C 180,E1 20105.07,E2 20105.07} C_VEL
LIN {X 0,Y 435.659,Z 689.575,A -85,B 0,C 180,E1 20100.784,E2 20100.784} C_VEL
LIN {X 0,Y 435.432,Z 694.209,A -85,B 0,C 180,E1 20100.404,E2 20100.404} C_VEL
LIN {X 0,Y 437.999,Z 716.976,A -85,B 0,C 180,E1 20099.85,E2 20099.85} C_VEL
LIN {X 0,Y 435.363,Z 894.336,A -85,B 0,C 180,E1 20096.91,E2 20096.91} C_VEL
LIN {X 0,Y 434.519,Z 913.075,A -85,B 0,C 180,E1 20096.367,E2 20096.367} C_VEL
LIN {X 0,Y 433.398,Z 931.27,A -85,B 0,C 180,E1 20095.594,E2 20095.594} C_VEL
LIN {X 0,Y 432.138,Z 948.874,A -85,B 0,C 180,E1 20094.591,E2 20094.591} C_VEL
LIN {X 0,Y 430.685,Z 966.345,A -85,B 0,C 180,E1 20093.318,E2 20093.318} C_VEL
LIN {X 0,Y 429.287,Z 982.221,A -85,B 0,C 180,E1 20091.88,E2 20091.88} C_VEL
LIN {X 0,Y 427.972,Z 997.187,A -85,B 0,C 180,E1 20090.229,E2 20090.229} C_VEL
LIN {X 0,Y 426.812,Z 1010.748,A -85,B 0,C 180,E1 20088.421,E2 20088.421} C_VEL
LIN {X 0,Y 425.803,Z 1023.517,A -85,B 0,C 180,E1 20086.367,E2 20086.367} C_VEL
LIN {X 0,Y 425.081,Z 1034.77,A -85,B 0,C 180,E1 20084.16,E2 20084.16} C_VEL
LIN {X 0,Y 424.612,Z 1044.394,A -85,B 0,C 180,E1 20081.822,E2 20081.822} C_VEL
LIN {X 0,Y 424.417,Z 1051.996,A -85,B 0,C 180,E1 20079.492,E2 20079.492} C_VEL
LIN {X 0,Y 424.374,Z 1057.783,A -85,B 0,C 180,E1 20077.174,E2 20077.174} C_VEL
LIN {X 0,Y 424.422,Z 1061.985,A -85,B 0,C 180,E1 20074.791,E2 20074.791} C_VEL
LIN {X 0,Y 424.498,Z 1064.476,A -85,B 0,C 180,E1 20072.43,E2 20072.43} C_VEL
LIN {X 0,Y 424.546,Z 1065.319,A -85,B 0,C 180,E1 20070,E2 20070} C_VEL
LIN {X 0,Y 424.504,Z 1064.424,A -85,B 0,C 180,E1 20067.57,E2 20067.57} C_VEL
LIN {X 0,Y 424.43,Z 1061.789,A -85,B 0,C 180,E1 20065.135,E2 20065.135} C_VEL
LIN {X 0,Y 424.39,Z 1057.365,A -85,B 0,C 180,E1 20062.689,E2 20062.689} C_VEL
LIN {X 0,Y 424.44,Z 1051.045,A -85,B 0,C 180,E1 20060.235,E2 20060.235} C_VEL
LIN {X 0,Y 424.661,Z 1043.172,A -85,B 0,C 180,E1 20057.904,E2 20057.904} C_VEL
LIN {X 0,Y 425.122,Z 1033.844,A -85,B 0,C 180,E1 20055.695,E2 20055.695} C_VEL
LIN {X 0,Y 425.856,Z 1022.438,A -85,B 0,C 180,E1 20053.495,E2 20053.495} C_VEL
LIN {X 0,Y 426.888,Z 1009.412,A -85,B 0,C 180,E1 20051.426,E2 20051.426} C_VEL
LIN {X 0,Y 428.088,Z 995.518,A -85,B 0,C 180,E1 20049.594,E2 20049.594} C_VEL
LIN {X 0,Y 429.461,Z 980.096,A -85,B 0,C 180,E1 20047.912,E2 20047.912} C_VEL
LIN {X 0,Y 430.911,Z 964.011,A -85,B 0,C 180,E1 20046.478,E2 20046.478} C_VEL
LIN {X 0,Y 432.349,Z 946.974,A -85,B 0,C 180,E1 20045.255,E2 20045.255} C_VEL
LIN {X 0,Y 433.63,Z 929.553,A -85,B 0,C 180,E1 20044.274,E2 20044.274} C_VEL
LIN {X 0,Y 434.774,Z 911.228,A -85,B 0,C 180,E1 20043.508,E2 20043.508} C_VEL
LIN {X 0,Y 435.638,Z 892.106,A -85,B 0,C 180,E1 20042.971,E2 20042.971} C_VEL
LIN {X 0,Y 438.228,Z 714.128,A -85,B 0,C 180,E1 20039.982,E2 20039.982} C_VEL
LIN {X 0,Y 435.812,Z 693.627,A -85,B 0,C 180,E1 20039.42,E2 20039.42} C_VEL
LIN {X 0,Y 439.95,Z 650.956,A -85,B 0,C 180,E1 20035.306,E2 20035.306} C_VEL
LIN {X 0,Y 440.515,Z 644.999,A -85,B 0,C 180,E1 20034.714,E2 20034.714} C_VEL
LIN {X 0,Y 434.908,Z 627.911,A -85,B 0,C 180,E1 20032.266,E2 20032.266} C_VEL
LIN {X 0,Y 429.15,Z 612.631,A -85,B 0,C 180,E1 20029.807,E2 20029.807} C_VEL
LIN {X 0,Y 425.347,Z 603.018,A -85,B 0,C 180,E1 20028.06,E2 20028.06} C_VEL
LIN {X 0,Y 425.301,Z 602.814,A -85,B 0,C 180,E1 20024.285,E2 20024.285} C_VEL
LIN {X 0,Y 425.27,Z 602.823,A -85,B 0,C 180,E1 20020.588,E2 20020.588} C_VEL
LIN {X 0,Y 425.267,Z 602.825,A -85,B 0,C 180,E1 20016.837,E2 20016.837} C_VEL
LIN {X 0,Y 425.298,Z 602.821,A -85,B 0,C 180,E1 20013.181,E2 20013.181} C_VEL
LIN {X 0,Y 425.33,Z 602.819,A -85,B 0,C 180,E1 20009.427,E2 20009.427} C_VEL
LIN {X 0,Y 425.301,Z 602.82,A -85,B 0,C 180,E1 20005.631,E2 20005.631} C_VEL
LIN {X 0,Y 425.272,Z 602.821,A -85,B 0,C 180,E1 20001.952,E2 20001.952} C_VEL
LIN {X 0,Y 425.271,Z 602.815,A -85,B 0,C 180,E1 19998.08,E2 19998.08} C_VEL
LIN {X 0,Y 425.292,Z 602.805,A -85,B 0,C 180,E1 19994.393,E2 19994.393} C_VEL
LIN {X 0,Y 425.318,Z 602.81,A -85,B 0,C 180,E1 19990.686,E2 19990.686} C_VEL
LIN {X 0,Y 425.306,Z 602.818,A -85,B 0,C 180,E1 19986.886,E2 19986.886} C_VEL
LIN {X 0,Y 425.281,Z 602.818,A -85,B 0,C 180,E1 19983.099,E2 19983.099} C_VEL
LIN {X 0,Y 425.278,Z 602.809,A -85,B 0,C 180,E1 19979.326,E2 19979.326} C_VEL
LIN {X 0,Y 425.294,Z 602.805,A -85,B 0,C 180,E1 19975.55,E2 19975.55} C_VEL
LIN {X 0,Y 425.32,Z 602.809,A -85,B 0,C 180,E1 19971.755,E2 19971.755} C_VEL
LIN {X 0,Y 425.316,Z 602.818,A -85,B 0,C 180,E1 19967.923,E2 19967.923} C_VEL
LIN {X 0,Y 425.296,Z 602.82,A -85,B 0,C 180,E1 19964.174,E2 19964.174} C_VEL
LIN {X 0,Y 425.288,Z 602.82,A -85,B 0,C 180,E1 19960.354,E2 19960.354} C_VEL
LIN {X 0,Y 425.29,Z 602.812,A -85,B 0,C 180,E1 19956.476,E2 19956.476} C_VEL
LIN {X 0,Y 425.312,Z 602.813,A -85,B 0,C 180,E1 19952.702,E2 19952.702} C_VEL
LIN {X 0,Y 425.322,Z 602.815,A -85,B 0,C 180,E1 19948.837,E2 19948.837} C_VEL
LIN {X 0,Y 425.354,Z 603.13,A -85,B 0,C 180,E1 19947.382,E2 19947.382} C_VEL
LIN {X 0,Y 429.974,Z 616.788,A -85,B 0,C 180,E1 19944.454,E2 19944.454} C_VEL
LIN {X 0,Y 434.389,Z 631.912,A -85,B 0,C 180,E1 19941.499,E2 19941.499} C_VEL
LIN {X 0,Y 436.123,Z 639.185,A -85,B 0,C 180,E1 19940.177,E2 19940.177} C_VEL
LIN {X 0,Y 433.371,Z 667.438,A -85,B 0,C 180,E1 19936.041,E2 19936.041} C_VEL
LIN {X 0,Y 430.995,Z 696.186,A -85,B 0,C 180,E1 19931.923,E2 19931.923} C_VEL
LIN {X 0,Y 430.187,Z 707.557,A -85,B 0,C 180,E1 19930.327,E2 19930.327} C_VEL
LIN {X 0,Y 431.555,Z 714.816,A -85,B 0,C 180,E1 19930.047,E2 19930.047} C_VEL
LIN {X 0,Y 434.408,Z 731.376,A -85,B 0,C 180,E1 19929.545,E2 19929.545} C_VEL
LIN {X 0,Y 432.599,Z 829.462,A -85,B 0,C 180,E1 19927.759,E2 19927.759} C_VEL
LIN {X 0,Y 432.111,Z 845.526,A -85,B 0,C 180,E1 19927.207,E2 19927.207} C_VEL
LIN {X 0,Y 431.41,Z 859.831,A -85,B 0,C 180,E1 19926.464,E2 19926.464} C_VEL
LIN {X 0,Y 430.529,Z 873.627,A -85,B 0,C 180,E1 19925.493,E2 19925.493} C_VEL
LIN {X 0,Y 429.49,Z 886.833,A -85,B 0,C 180,E1 19924.264,E2 19924.264} C_VEL
LIN {X 0,Y 428.523,Z 898.06,A -85,B 0,C 180,E1 19922.932,E2 19922.932} C_VEL
LIN {X 0,Y 427.502,Z 909.021,A -85,B 0,C 180,E1 19921.28,E2 19921.28} C_VEL
LIN {X 0,Y 426.604,Z 918.179,A -85,B 0,C 180,E1 19919.485,E2 19919.485} C_VEL
LIN {X 0,Y 426.152,Z 922.892,A -85,B 0,C 180,E1 19918.336,E2 19918.336} C_VEL
LIN {X 0,Y 424.878,Z 926.34,A -85,B 0,C 180,E1 19917.41,E2 19917.41} C_VEL
LIN {X 0,Y 420.083,Z 931.978,A -85,B 0,C 180,E1 19915.712,E2 19915.712} C_VEL
LIN {X 0,Y 417.623,Z 934.783,A -85,B 0,C 180,E1 19914.521,E2 19914.521} C_VEL
LIN {X 0,Y 417.27,Z 935.629,A -85,B 0,C 180,E1 19914.003,E2 19914.003} C_VEL
LIN {X 0,Y 417.062,Z 937.973,A -85,B 0,C 180,E1 19911.814,E2 19911.814} C_VEL
LIN {X 0,Y 416.995,Z 938.463,A -85,B 0,C 180,E1 19909.76,E2 19909.76} C_VEL
LIN {X 0,Y 417.04,Z 937.23,A -85,B 0,C 180,E1 19907.583,E2 19907.583} C_VEL
LIN {X 0,Y 417.22,Z 934.106,A -85,B 0,C 180,E1 19905.427,E2 19905.427} C_VEL
LIN {X 0,Y 417.559,Z 929.463,A -85,B 0,C 180,E1 19903.431,E2 19903.431} C_VEL
LIN {X 0,Y 418.13,Z 922.563,A -85,B 0,C 180,E1 19901.355,E2 19901.355} C_VEL
LIN {X 0,Y 418.881,Z 914.126,A -85,B 0,C 180,E1 19899.48,E2 19899.48} C_VEL
LIN {X 0,Y 419.768,Z 904.415,A -85,B 0,C 180,E1 19897.803,E2 19897.803} C_VEL
LIN {X 0,Y 420.77,Z 892.595,A -85,B 0,C 180,E1 19896.207,E2 19896.207} C_VEL
LIN {X 0,Y 421.747,Z 880.062,A -85,B 0,C 180,E1 19894.896,E2 19894.896} C_VEL
LIN {X 0,Y 422.629,Z 867.488,A -85,B 0,C 180,E1 19893.866,E2 19893.866} C_VEL
LIN {X 0,Y 423.45,Z 852.388,A -85,B 0,C 180,E1 19892.94,E2 19892.94} C_VEL
LIN {X 0,Y 424.019,Z 837.161,A -85,B 0,C 180,E1 19892.293,E2 19892.293} C_VEL
LIN {X 0,Y 424.343,Z 821.294,A -85,B 0,C 180,E1 19891.882,E2 19891.882} C_VEL
LIN {X 0,Y 425.665,Z 729.672,A -85,B 0,C 180,E1 19890.252,E2 19890.252} C_VEL
LIN {X 0,Y 421.795,Z 707.666,A -85,B 0,C 180,E1 19889.592,E2 19889.592} C_VEL
LIN {X 0,Y 423.83,Z 678.865,A -85,B 0,C 180,E1 19885.535,E2 19885.535} C_VEL
LIN {X 0,Y 426.151,Z 650.764,A -85,B 0,C 180,E1 19881.499,E2 19881.499} C_VEL
LIN {X 0,Y 427.242,Z 638.706,A -85,B 0,C 180,E1 19879.755,E2 19879.755} C_VEL
LIN {X 0,Y 422.476,Z 620.908,A -85,B 0,C 180,E1 19876.583,E2 19876.583} C_VEL
LIN {X 0,Y 417.391,Z 603.925,A -85,B 0,C 180,E1 19873.347,E2 19873.347} C_VEL
LIN {X 0,Y 417.37,Z 603.804,A -85,B 0,C 180,E1 19869.38,E2 19869.38} C_VEL
LIN {X 0,Y 417.359,Z 603.769,A -85,B 0,C 180,E1 19865.515,E2 19865.515} C_VEL
LIN {X 0,Y 417.374,Z 603.801,A -85,B 0,C 180,E1 19861.684,E2 19861.684} C_VEL
LIN {X 0,Y 417.375,Z 603.768,A -85,B 0,C 180,E1 19857.871,E2 19857.871} C_VEL
LIN {X 0,Y 417.378,Z 603.804,A -85,B 0,C 180,E1 19854.061,E2 19854.061} C_VEL
LIN {X 0,Y 417.382,Z 603.809,A -85,B 0,C 180,E1 19850.237,E2 19850.237} C_VEL
LIN {X 0,Y 417.364,Z 603.791,A -85,B 0,C 180,E1 19846.344,E2 19846.344} C_VEL
LIN {X 0,Y 417.357,Z 603.804,A -85,B 0,C 180,E1 19842.449,E2 19842.449} C_VEL
LIN {X 0,Y 417.356,Z 603.804,A -85,B 0,C 180,E1 19838.527,E2 19838.527} C_VEL
LIN {X 0,Y 417.369,Z 603.789,A -85,B 0,C 180,E1 19834.744,E2 19834.744} C_VEL
LIN {X 0,Y 417.387,Z 603.804,A -85,B 0,C 180,E1 19830.84,E2 19830.84} C_VEL
LIN {X 0,Y 417.381,Z 603.781,A -85,B 0,C 180,E1 19826.921,E2 19826.921} C_VEL
LIN {X 0,Y 417.381,Z 603.804,A -85,B 0,C 180,E1 19822.984,E2 19822.984} C_VEL
LIN {X 0,Y 417.355,Z 603.791,A -85,B 0,C 180,E1 19819.161,E2 19819.161} C_VEL
LIN {X 0,Y 417.346,Z 603.798,A -85,B 0,C 180,E1 19815.28,E2 19815.28} C_VEL
LIN {X 0,Y 417.345,Z 603.804,A -85,B 0,C 180,E1 19811.33,E2 19811.33} C_VEL
LIN {X 0,Y 417.353,Z 603.791,A -85,B 0,C 180,E1 19807.433,E2 19807.433} C_VEL
LIN {X 0,Y 417.374,Z 603.801,A -85,B 0,C 180,E1 19803.709,E2 19803.709} C_VEL
LIN {X 0,Y 417.387,Z 603.78,A -85,B 0,C 180,E1 19799.863,E2 19799.863} C_VEL
LIN {X 0,Y 417.366,Z 603.81,A -85,B 0,C 180,E1 19796.017,E2 19796.017} C_VEL
LIN {X 0,Y 417.334,Z 603.785,A -85,B 0,C 180,E1 19792.29,E2 19792.29} C_VEL
LIN {X 0,Y 417.337,Z 603.81,A -85,B 0,C 180,E1 19788.39,E2 19788.39} C_VEL
LIN {X 0,Y 417.348,Z 603.797,A -85,B 0,C 180,E1 19784.578,E2 19784.578} C_VEL
LIN {X 0,Y 417.376,Z 603.798,A -85,B 0,C 180,E1 19780.841,E2 19780.841} C_VEL
LIN {X 0,Y 417.389,Z 603.807,A -85,B 0,C 180,E1 19777.017,E2 19777.017} C_VEL
LIN {X 0,Y 417.364,Z 603.796,A -85,B 0,C 180,E1 19773.078,E2 19773.078} C_VEL
LIN {X 0,Y 417.327,Z 603.803,A -85,B 0,C 180,E1 19769.475,E2 19769.475} C_VEL
LIN {X 0,Y 417.336,Z 603.806,A -85,B 0,C 180,E1 19765.736,E2 19765.736} C_VEL
LIN {X 0,Y 417.369,Z 603.8,A -85,B 0,C 180,E1 19761.999,E2 19761.999} C_VEL
LIN {X 0,Y 417.385,Z 603.799,A -85,B 0,C 180,E1 19758.161,E2 19758.161} C_VEL
LIN {X 0,Y 417.368,Z 603.811,A -85,B 0,C 180,E1 19754.251,E2 19754.251} C_VEL
LIN {X 0,Y 417.387,Z 604.019,A -85,B 0,C 180,E1 19751.497,E2 19751.497} C_VEL
LIN {X 0,Y 421.125,Z 614.398,A -85,B 0,C 180,E1 19749.871,E2 19749.871} C_VEL
LIN {X 0,Y 428.424,Z 634.901,A -85,B 0,C 180,E1 19746.934,E2 19746.934} C_VEL
LIN {X 0,Y 432.285,Z 647.05,A -85,B 0,C 180,E1 19745.327,E2 19745.327} C_VEL
LIN {X 0,Y 428.06,Z 692.168,A -85,B 0,C 180,E1 19740.993,E2 19740.993} C_VEL
LIN {X 0,Y 428.075,Z 694.851,A -85,B 0,C 180,E1 19740.825,E2 19740.825} C_VEL
LIN {X 0,Y 430.654,Z 717.989,A -85,B 0,C 180,E1 19740.258,E2 19740.258} C_VEL
LIN {X 0,Y 427.896,Z 893.625,A -85,B 0,C 180,E1 19737.3,E2 19737.3} C_VEL
LIN {X 0,Y 427.019,Z 912.263,A -85,B 0,C 180,E1 19736.754,E2 19736.754} C_VEL
LIN {X 0,Y 425.851,Z 930.474,A -85,B 0,C 180,E1 19735.969,E2 19735.969} C_VEL
LIN {X 0,Y 424.498,Z 948.379,A -85,B 0,C 180,E1 19734.93,E2 19734.93} C_VEL
LIN {X 0,Y 423.04,Z 965.103,A -85,B 0,C 180,E1 19733.691,E2 19733.691} C_VEL
LIN {X 0,Y 421.562,Z 981.015,A -85,B 0,C 180,E1 19732.231,E2 19732.231} C_VEL
LIN {X 0,Y 420.176,Z 996.033,A -85,B 0,C 180,E1 19730.549,E2 19730.549} C_VEL
LIN {X 0,Y 418.916,Z 1010.107,A -85,B 0,C 180,E1 19728.64,E2 19728.64} C_VEL
LIN {X 0,Y 417.864,Z 1022.854,A -85,B 0,C 180,E1 19726.544,E2 19726.544} C_VEL
LIN {X 0,Y 417.115,Z 1034.029,A -85,B 0,C 180,E1 19724.294,E2 19724.294} C_VEL
LIN {X 0,Y 416.657,Z 1043.092,A -85,B 0,C 180,E1 19722.051,E2 19722.051} C_VEL
LIN {X 0,Y 416.455,Z 1050.732,A -85,B 0,C 180,E1 19719.675,E2 19719.675} C_VEL
LIN {X 0,Y 416.426,Z 1056.55,A -85,B 0,C 180,E1 19717.311,E2 19717.311} C_VEL
LIN {X 0,Y 416.486,Z 1060.706,A -85,B 0,C 180,E1 19714.937,E2 19714.937} C_VEL
LIN {X 0,Y 416.58,Z 1063.278,A -85,B 0,C 180,E1 19712.476,E2 19712.476} C_VEL
LIN {X 0,Y 416.635,Z 1064.126,A -85,B 0,C 180,E1 19710,E2 19710} C_VEL
LIN {X 0,Y 416.586,Z 1063.227,A -85,B 0,C 180,E1 19707.524,E2 19707.524} C_VEL
LIN {X 0,Y 416.498,Z 1060.58,A -85,B 0,C 180,E1 19705.042,E2 19705.042} C_VEL
LIN {X 0,Y 416.44,Z 1056.137,A -85,B 0,C 180,E1 19702.551,E2 19702.551} C_VEL
LIN {X 0,Y 416.477,Z 1049.779,A -85,B 0,C 180,E1 19700.046,E2 19700.046} C_VEL
LIN {X 0,Y 416.709,Z 1041.866,A -85,B 0,C 180,E1 19697.67,E2 19697.67} C_VEL
LIN {X 0,Y 417.233,Z 1031.883,A -85,B 0,C 180,E1 19695.285,E2 19695.285} C_VEL
LIN {X 0,Y 418.019,Z 1020.603,A -85,B 0,C 180,E1 19693.089,E2 19693.089} C_VEL
LIN {X 0,Y 419.084,Z 1008.038,A -85,B 0,C 180,E1 19691.067,E2 19691.067} C_VEL
LIN {X 0,Y 420.386,Z 993.925,A -85,B 0,C 180,E1 19689.183,E2 19689.183} C_VEL
LIN {X 0,Y 421.836,Z 978.591,A -85,B 0,C 180,E1 19687.493,E2 19687.493} C_VEL
LIN {X 0,Y 423.387,Z 962.375,A -85,B 0,C 180,E1 19686.034,E2 19686.034} C_VEL
LIN {X 0,Y 424.906,Z 945.168,A -85,B 0,C 180,E1 19684.791,E2 19684.791} C_VEL
LIN {X 0,Y 426.338,Z 926.864,A -85,B 0,C 180,E1 19683.764,E2 19683.764} C_VEL
LIN {X 0,Y 427.526,Z 908.192,A -85,B 0,C 180,E1 19683.003,E2 19683.003} C_VEL
LIN {X 0,Y 428.351,Z 889.418,A -85,B 0,C 180,E1 19682.498,E2 19682.498} C_VEL
LIN {X 0,Y 431.064,Z 715.155,A -85,B 0,C 180,E1 19679.524,E2 19679.524} C_VEL
LIN {X 0,Y 428.577,Z 693.8,A -85,B 0,C 180,E1 19678.924,E2 19678.924} C_VEL
LIN {X 0,Y 433.012,Z 651.331,A -85,B 0,C 180,E1 19674.741,E2 19674.741} C_VEL
LIN {X 0,Y 433.231,Z 647.405,A -85,B 0,C 180,E1 19674.329,E2 19674.329} C_VEL
LIN {X 0,Y 427.867,Z 631.048,A -85,B 0,C 180,E1 19671.908,E2 19671.908} C_VEL
LIN {X 0,Y 422.305,Z 616.274,A -85,B 0,C 180,E1 19669.465,E2 19669.465} C_VEL
LIN {X 0,Y 418.133,Z 606.402,A -85,B 0,C 180,E1 19667.637,E2 19667.637} C_VEL
LIN {X 0,Y 417.348,Z 603.972,A -85,B 0,C 180,E1 19667.126,E2 19667.126} C_VEL
LIN {X 0,Y 417.346,Z 603.808,A -85,B 0,C 180,E1 19663.439,E2 19663.439} C_VEL
LIN {X 0,Y 417.39,Z 603.807,A -85,B 0,C 180,E1 19659.74,E2 19659.74} C_VEL
LIN {X 0,Y 417.364,Z 603.802,A -85,B 0,C 180,E1 19655.93,E2 19655.93} C_VEL
LIN {X 0,Y 417.34,Z 603.802,A -85,B 0,C 180,E1 19652.131,E2 19652.131} C_VEL
LIN {X 0,Y 417.329,Z 603.803,A -85,B 0,C 180,E1 19648.444,E2 19648.444} C_VEL
LIN {X 0,Y 417.342,Z 603.804,A -85,B 0,C 180,E1 19644.637,E2 19644.637} C_VEL
LIN {X 0,Y 417.374,Z 603.808,A -85,B 0,C 180,E1 19640.888,E2 19640.888} C_VEL
LIN {X 0,Y 417.38,Z 603.805,A -85,B 0,C 180,E1 19636.993,E2 19636.993} C_VEL
LIN {X 0,Y 417.36,Z 603.8,A -85,B 0,C 180,E1 19633.155,E2 19633.155} C_VEL
LIN {X 0,Y 417.34,Z 603.791,A -85,B 0,C 180,E1 19629.376,E2 19629.376} C_VEL
LIN {X 0,Y 417.337,Z 603.8,A -85,B 0,C 180,E1 19625.637,E2 19625.637} C_VEL
LIN {X 0,Y 417.352,Z 603.809,A -85,B 0,C 180,E1 19621.784,E2 19621.784} C_VEL
LIN {X 0,Y 417.379,Z 603.803,A -85,B 0,C 180,E1 19618.078,E2 19618.078} C_VEL
LIN {X 0,Y 417.382,Z 603.795,A -85,B 0,C 180,E1 19614.087,E2 19614.087} C_VEL
LIN {X 0,Y 417.357,Z 603.792,A -85,B 0,C 180,E1 19610.346,E2 19610.346} C_VEL
LIN {X 0,Y 417.344,Z 603.795,A -85,B 0,C 180,E1 19606.562,E2 19606.562} C_VEL
LIN {X 0,Y 417.348,Z 603.798,A -85,B 0,C 180,E1 19602.718,E2 19602.718} C_VEL
LIN {X 0,Y 417.369,Z 603.798,A -85,B 0,C 180,E1 19598.94,E2 19598.94} C_VEL
LIN {X 0,Y 417.38,Z 603.803,A -85,B 0,C 180,E1 19595.063,E2 19595.063} C_VEL
LIN {X 0,Y 417.386,Z 603.803,A -85,B 0,C 180,E1 19591.216,E2 19591.216} C_VEL
LIN {X 0,Y 417.397,Z 604.073,A -85,B 0,C 180,E1 19588.259,E2 19588.259} C_VEL
LIN {X 0,Y 422.142,Z 617.805,A -85,B 0,C 180,E1 19585.192,E2 19585.192} C_VEL
LIN {X 0,Y 426.459,Z 632.219,A -85,B 0,C 180,E1 19582.27,E2 19582.27} C_VEL
LIN {X 0,Y 428.812,Z 642.152,A -85,B 0,C 180,E1 19580.41,E2 19580.41} C_VEL
LIN {X 0,Y 425.968,Z 669.87,A -85,B 0,C 180,E1 19576.299,E2 19576.299} C_VEL
LIN {X 0,Y 423.428,Z 698.579,A -85,B 0,C 180,E1 19572.115,E2 19572.115} C_VEL
LIN {X 0,Y 422.792,Z 707.929,A -85,B 0,C 180,E1 19570.819,E2 19570.819} C_VEL
LIN {X 0,Y 427.266,Z 732.076,A -85,B 0,C 180,E1 19570.018,E2 19570.018} C_VEL
LIN {X 0,Y 425.338,Z 830.133,A -85,B 0,C 180,E1 19568.199,E2 19568.199} C_VEL
LIN {X 0,Y 424.808,Z 846.532,A -85,B 0,C 180,E1 19567.624,E2 19567.624} C_VEL
LIN {X 0,Y 424.068,Z 860.693,A -85,B 0,C 180,E1 19566.874,E2 19566.874} C_VEL
LIN {X 0,Y 423.092,Z 874.975,A -85,B 0,C 180,E1 19565.846,E2 19565.846} C_VEL
LIN {X 0,Y 421.947,Z 888.594,A -85,B 0,C 180,E1 19564.545,E2 19564.545} C_VEL
LIN {X 0,Y 420.863,Z 900.131,A -85,B 0,C 180,E1 19563.122,E2 19563.122} C_VEL
LIN {X 0,Y 419.815,Z 910.528,A -85,B 0,C 180,E1 19561.5,E2 19561.5} C_VEL
LIN {X 0,Y 418.826,Z 919.839,A -85,B 0,C 180,E1 19559.615,E2 19559.615} C_VEL
LIN {X 0,Y 418.105,Z 926.761,A -85,B 0,C 180,E1 19557.77,E2 19557.77} C_VEL
LIN {X 0,Y 417.554,Z 932.483,A -85,B 0,C 180,E1 19555.684,E2 19555.684} C_VEL
LIN {X 0,Y 417.27,Z 935.629,A -85,B 0,C 180,E1 19554.003,E2 19554.003} C_VEL
LIN {X 0,Y 416.156,Z 937.131,A -85,B 0,C 180,E1 19552.964,E2 19552.964} C_VEL
LIN {X 0,Y 411.807,Z 939.142,A -85,B 0,C 180,E1 19551.143,E2 19551.143} C_VEL
LIN {X 0,Y 409.356,Z 939.636,A -85,B 0,C 180,E1 19549.785,E2 19549.785} C_VEL
LIN {X 0,Y 409.082,Z 939.537,A -85,B 0,C 180,E1 19549.241,E2 19549.241} C_VEL
LIN {X 0,Y 409.157,Z 937.85,A -85,B 0,C 180,E1 19547.052,E2 19547.052} C_VEL
LIN {X 0,Y 409.379,Z 934.638,A -85,B 0,C 180,E1 19545.004,E2 19545.004} C_VEL
LIN {X 0,Y 409.806,Z 929.235,A -85,B 0,C 180,E1 19542.828,E2 19542.828} C_VEL
LIN {X 0,Y 410.391,Z 922.672,A -85,B 0,C 180,E1 19540.93,E2 19540.93} C_VEL
LIN {X 0,Y 411.191,Z 914.344,A -85,B 0,C 180,E1 19539.094,E2 19539.094} C_VEL
LIN {X 0,Y 412.145,Z 904.361,A -85,B 0,C 180,E1 19537.387,E2 19537.387} C_VEL
LIN {X 0,Y 413.127,Z 893.325,A -85,B 0,C 180,E1 19535.891,E2 19535.891} C_VEL
LIN {X 0,Y 414.218,Z 880.057,A -85,B 0,C 180,E1 19534.494,E2 19534.494} C_VEL
LIN {X 0,Y 415.133,Z 867.258,A -85,B 0,C 180,E1 19533.452,E2 19533.452} C_VEL
LIN {X 0,Y 415.967,Z 852.579,A -85,B 0,C 180,E1 19532.548,E2 19532.548} C_VEL
LIN {X 0,Y 416.567,Z 836.83,A -85,B 0,C 180,E1 19531.882,E2 19531.882} C_VEL
LIN {X 0,Y 416.891,Z 820.87,A -85,B 0,C 180,E1 19531.477,E2 19531.477} C_VEL
LIN {X 0,Y 418.279,Z 730.736,A -85,B 0,C 180,E1 19529.844,E2 19529.844} C_VEL
LIN {X 0,Y 414.258,Z 708.055,A -85,B 0,C 180,E1 19529.17,E2 19529.17} C_VEL
LIN {X 0,Y 414.437,Z 703.716,A -85,B 0,C 180,E1 19528.617,E2 19528.617} C_VEL
LIN {X 0,Y 416.678,Z 675.141,A -85,B 0,C 180,E1 19524.492,E2 19524.492} C_VEL
LIN {X 0,Y 419.191,Z 647,A -85,B 0,C 180,E1 19520.388,E2 19520.388} C_VEL
LIN {X 0,Y 419.61,Z 640.565,A -85,B 0,C 180,E1 19519.427,E2 19519.427} C_VEL
LIN {X 0,Y 414.815,Z 622.764,A -85,B 0,C 180,E1 19516.194,E2 19516.194} C_VEL
LIN {X 0,Y 409.969,Z 606.828,A -85,B 0,C 180,E1 19513.128,E2 19513.128} C_VEL
LIN {X 0,Y 409.447,Z 604.868,A -85,B 0,C 180,E1 19512.667,E2 19512.667} C_VEL
LIN {X 0,Y 409.439,Z 604.797,A -85,B 0,C 180,E1 19508.662,E2 19508.662} C_VEL
LIN {X 0,Y 409.436,Z 604.766,A -85,B 0,C 180,E1 19504.7,E2 19504.7} C_VEL
LIN {X 0,Y 409.438,Z 604.765,A -85,B 0,C 180,E1 19500.764,E2 19500.764} C_VEL
LIN {X 0,Y 409.425,Z 604.778,A -85,B 0,C 180,E1 19496.836,E2 19496.836} C_VEL
LIN {X 0,Y 409.42,Z 604.787,A -85,B 0,C 180,E1 19492.899,E2 19492.899} C_VEL
LIN {X 0,Y 409.423,Z 604.797,A -85,B 0,C 180,E1 19488.933,E2 19488.933} C_VEL
LIN {X 0,Y 409.432,Z 604.792,A -85,B 0,C 180,E1 19485.089,E2 19485.089} C_VEL
LIN {X 0,Y 409.446,Z 604.77,A -85,B 0,C 180,E1 19481.224,E2 19481.224} C_VEL
LIN {X 0,Y 409.442,Z 604.794,A -85,B 0,C 180,E1 19477.241,E2 19477.241} C_VEL
LIN {X 0,Y 409.44,Z 604.771,A -85,B 0,C 180,E1 19473.33,E2 19473.33} C_VEL
LIN {X 0,Y 409.436,Z 604.797,A -85,B 0,C 180,E1 19469.397,E2 19469.397} C_VEL
LIN {X 0,Y 409.419,Z 604.768,A -85,B 0,C 180,E1 19465.456,E2 19465.456} C_VEL
LIN {X 0,Y 409.41,Z 604.798,A -85,B 0,C 180,E1 19461.64,E2 19461.64} C_VEL
LIN {X 0,Y 409.409,Z 604.766,A -85,B 0,C 180,E1 19457.736,E2 19457.736} C_VEL
LIN {X 0,Y 409.426,Z 604.794,A -85,B 0,C 180,E1 19453.847,E2 19453.847} C_VEL
LIN {X 0,Y 409.435,Z 604.769,A -85,B 0,C 180,E1 19449.985,E2 19449.985} C_VEL
LIN {X 0,Y 409.446,Z 604.788,A -85,B 0,C 180,E1 19446.168,E2 19446.168} C_VEL
LIN {X 0,Y 409.427,Z 604.778,A -85,B 0,C 180,E1 19442.24,E2 19442.24} C_VEL
LIN {X 0,Y 409.403,Z 604.787,A -85,B 0,C 180,E1 19438.461,E2 19438.461} C_VEL
LIN {X 0,Y 409.399,Z 604.794,A -85,B 0,C 180,E1 19434.675,E2 19434.675} C_VEL
LIN {X 0,Y 409.413,Z 604.79,A -85,B 0,C 180,E1 19430.866,E2 19430.866} C_VEL
LIN {X 0,Y 409.434,Z 604.783,A -85,B 0,C 180,E1 19427.005,E2 19427.005} C_VEL
LIN {X 0,Y 409.445,Z 604.797,A -85,B 0,C 180,E1 19423.107,E2 19423.107} C_VEL
LIN {X 0,Y 409.442,Z 604.778,A -85,B 0,C 180,E1 19419.113,E2 19419.113} C_VEL
